LIN {X 0,Y 210.125,Z 422.294,A -85,B 0,C 180,E1 -20903.58,E2 -20903.58} C_VEL
LIN {X 0,Y 207.725,Z 422.606,A -85,B 0,C 180,E1 -20905.677,E2 -20905.677} C_VEL
LIN {X 0,Y 206.757,Z 422.716,A -85,B 0,C 180,E1 -20907.307,E2 -20907.307} C_VEL
LIN {X 0,Y 206.709,Z 422.715,A -85,B 0,C 180,E1 -20907.858,E2 -20907.858} C_VEL
LIN {X 0,Y 206.696,Z 422.724,A -85,B 0,C 180,E1 -20912.958,E2 -20912.958} C_VEL
LIN {X 0,Y 206.724,Z 422.922,A -85,B 0,C 180,E1 -20915.32,E2 -20915.32} C_VEL
LIN {X 0,Y 206.934,Z 423.791,A -85,B 0,C 180,E1 -20915.862,E2 -20915.862} C_VEL
LIN {X 0,Y 207.388,Z 425.01,A -85,B 0,C 180,E1 -20916.372,E2 -20916.372} C_VEL
LIN {X 0,Y 209.51,Z 427.919,A -85,B 0,C 180,E1 -20917.883,E2 -20917.883} C_VEL
LIN {X 0,Y 211.221,Z 431.051,A -85,B 0,C 180,E1 -20919.212,E2 -20919.212} C_VEL
LIN {X 0,Y 211.934,Z 431.967,A -85,B 0,C 180,E1 -20919.67,E2 -20919.67} C_VEL
LIN {X 0,Y 217.278,Z 441.785,A -85,B 0,C 180,E1 -20923.342,E2 -20923.342} C_VEL
LIN {X 0,Y 222.7,Z 451.851,A -85,B 0,C 180,E1 -20926.539,E2 -20926.539} C_VEL
LIN {X 0,Y 223.952,Z 454.762,A -85,B 0,C 180,E1 -20927.32,E2 -20927.32} C_VEL
LIN {X 0,Y 227.39,Z 471.394,A -85,B 0,C 180,E1 -20930.595,E2 -20930.595} C_VEL
LIN {X 0,Y 227.539,Z 474.416,A -85,B 0,C 180,E1 -20931.074,E2 -20931.074} C_VEL
LIN {X 0,Y 226.465,Z 488.855,A -85,B 0,C 180,E1 -20932.939,E2 -20932.939} C_VEL
LIN {X 0,Y 229.261,Z 519.875,A -85,B 0,C 180,E1 -20934.642,E2 -20934.642} C_VEL
LIN {X 0,Y 230.377,Z 537.62,A -85,B 0,C 180,E1 -20935.498,E2 -20935.498} C_VEL
LIN {X 0,Y 227.64,Z 600.474,A -85,B 0,C 180,E1 -20937.362,E2 -20937.362} C_VEL
LIN {X 0,Y 226.564,Z 613.93,A -85,B 0,C 180,E1 -20937.977,E2 -20937.977} C_VEL
LIN {X 0,Y 224.9,Z 626.109,A -85,B 0,C 180,E1 -20938.83,E2 -20938.83} C_VEL
LIN {X 0,Y 222.978,Z 637.557,A -85,B 0,C 180,E1 -20939.976,E2 -20939.976} C_VEL
LIN {X 0,Y 220.64,Z 648.728,A -85,B 0,C 180,E1 -20941.458,E2 -20941.458} C_VEL
LIN {X 0,Y 217.804,Z 660.086,A -85,B 0,C 180,E1 -20943.403,E2 -20943.403} C_VEL
LIN {X 0,Y 215.262,Z 669.231,A -85,B 0,C 180,E1 -20945.4,E2 -20945.4} C_VEL
LIN {X 0,Y 212.776,Z 678.047,A -85,B 0,C 180,E1 -20947.847,E2 -20947.847} C_VEL
LIN {X 0,Y 210.351,Z 685.667,A -85,B 0,C 180,E1 -20950.481,E2 -20950.481} C_VEL
LIN {X 0,Y 208.205,Z 692.195,A -85,B 0,C 180,E1 -20953.326,E2 -20953.326} C_VEL
LIN {X 0,Y 206.629,Z 697.379,A -85,B 0,C 180,E1 -20956.226,E2 -20956.226} C_VEL
LIN {X 0,Y 205.499,Z 701.381,A -85,B 0,C 180,E1 -20959.158,E2 -20959.158} C_VEL
LIN {X 0,Y 204.766,Z 704.328,A -85,B 0,C 180,E1 -20962.109,E2 -20962.109} C_VEL
LIN {X 0,Y 204.411,Z 706.558,A -85,B 0,C 180,E1 -20965.613,E2 -20965.613} C_VEL
LIN {X 0,Y 204.367,Z 707.347,A -85,B 0,C 180,E1 -20968.029,E2 -20968.029} C_VEL
LIN {X 0,Y 204.421,Z 707.561,A -85,B 0,C 180,E1 -20970,E2 -20970} C_VEL
LIN {X 0,Y 204.394,Z 707.335,A -85,B 0,C 180,E1 -20971.97,E2 -20971.97} C_VEL
LIN {X 0,Y 204.439,Z 706.499,A -85,B 0,C 180,E1 -20974.487,E2 -20974.487} C_VEL
LIN {X 0,Y 204.77,Z 704.285,A -85,B 0,C 180,E1 -20977.891,E2 -20977.891} C_VEL
LIN {X 0,Y 205.5,Z 701.321,A -85,B 0,C 180,E1 -20980.842,E2 -20980.842} C_VEL
LIN {X 0,Y 206.632,Z 697.298,A -85,B 0,C 180,E1 -20983.773,E2 -20983.773} C_VEL
LIN {X 0,Y 208.571,Z 691.095,A -85,B 0,C 180,E1 -20987.148,E2 -20987.148} C_VEL
LIN {X 0,Y 210.742,Z 684.327,A -85,B 0,C 180,E1 -20989.988,E2 -20989.988} C_VEL
LIN {X 0,Y 213.138,Z 676.486,A -85,B 0,C 180,E1 -20992.591,E2 -20992.591} C_VEL
LIN {X 0,Y 215.796,Z 667.107,A -85,B 0,C 180,E1 -20995.048,E2 -20995.048} C_VEL
LIN {X 0,Y 218.722,Z 656.357,A -85,B 0,C 180,E1 -20997.25,E2 -20997.25} C_VEL
LIN {X 0,Y 221.283,Z 645.5,A -85,B 0,C 180,E1 -20998.969,E2 -20998.969} C_VEL
LIN {X 0,Y 221.982,Z 642.83,A -85,B 0,C 180,E1 -20999.389,E2 -20999.389} C_VEL
LIN {X 0,Y 227.16,Z 636.768,A -85,B 0,C 180,E1 -21001.732,E2 -21001.732} C_VEL
LIN {X 0,Y 234.125,Z 628.278,A -85,B 0,C 180,E1 -21004.252,E2 -21004.252} C_VEL
LIN {X 0,Y 241.939,Z 617.995,A -85,B 0,C 180,E1 -21006.548,E2 -21006.548} C_VEL
LIN {X 0,Y 249.222,Z 607.391,A -85,B 0,C 180,E1 -21008.345,E2 -21008.345} C_VEL
LIN {X 0,Y 256.826,Z 594.892,A -85,B 0,C 180,E1 -21009.985,E2 -21009.985} C_VEL
LIN {X 0,Y 263.198,Z 583.1,A -85,B 0,C 180,E1 -21011.138,E2 -21011.138} C_VEL
LIN {X 0,Y 269.507,Z 569.488,A -85,B 0,C 180,E1 -21012.182,E2 -21012.182} C_VEL
LIN {X 0,Y 274.93,Z 555.525,A -85,B 0,C 180,E1 -21013.012,E2 -21013.012} C_VEL
LIN {X 0,Y 278.395,Z 544.603,A -85,B 0,C 180,E1 -21013.614,E2 -21013.614} C_VEL
LIN {X 0,Y 280.825,Z 534.789,A -85,B 0,C 180,E1 -21014.437,E2 -21014.437} C_VEL
LIN {X 0,Y 283.081,Z 524.784,A -85,B 0,C 180,E1 -21015.548,E2 -21015.548} C_VEL
LIN {X 0,Y 283.658,Z 522.171,A -85,B 0,C 180,E1 -21017.163,E2 -21017.163} C_VEL
LIN {X 0,Y 284.036,Z 521.4,A -85,B 0,C 180,E1 -21018.01,E2 -21018.01} C_VEL
LIN {X 0,Y 280.282,Z 536.18,A -85,B 0,C 180,E1 -21018.966,E2 -21018.966} C_VEL
LIN {X 0,Y 276.118,Z 548.931,A -85,B 0,C 180,E1 -21020.007,E2 -21020.007} C_VEL
LIN {X 0,Y 271.63,Z 559.907,A -85,B 0,C 180,E1 -21021.139,E2 -21021.139} C_VEL
LIN {X 0,Y 266.158,Z 571.085,A -85,B 0,C 180,E1 -21022.604,E2 -21022.604} C_VEL
LIN {X 0,Y 259.706,Z 582.081,A -85,B 0,C 180,E1 -21024.421,E2 -21024.421} C_VEL
LIN {X 0,Y 253.474,Z 591.011,A -85,B 0,C 180,E1 -21026.321,E2 -21026.321} C_VEL
LIN {X 0,Y 247.643,Z 598.282,A -85,B 0,C 180,E1 -21028.33,E2 -21028.33} C_VEL
LIN {X 0,Y 242.063,Z 604.273,A -85,B 0,C 180,E1 -21030.424,E2 -21030.424} C_VEL
LIN {X 0,Y 236.808,Z 609.042,A -85,B 0,C 180,E1 -21032.612,E2 -21032.612} C_VEL
LIN {X 0,Y 231.875,Z 612.783,A -85,B 0,C 180,E1 -21034.892,E2 -21034.892} C_VEL
LIN {X 0,Y 228.801,Z 614.725,A -85,B 0,C 180,E1 -21036.465,E2 -21036.465} C_VEL
LIN {X 0,Y 225.905,Z 616.243,A -85,B 0,C 180,E1 -21038.079,E2 -21038.079} C_VEL
LIN {X 0,Y 220.673,Z 618.05,A -85,B 0,C 180,E1 -21041.429,E2 -21041.429} C_VEL
LIN {X 0,Y 216.251,Z 618.267,A -85,B 0,C 180,E1 -21044.93,E2 -21044.93} C_VEL
LIN {X 0,Y 214.361,Z 617.789,A -85,B 0,C 180,E1 -21046.732,E2 -21046.732} C_VEL
LIN {X 0,Y 211.13,Z 615.597,A -85,B 0,C 180,E1 -21050.419,E2 -21050.419} C_VEL
LIN {X 0,Y 209.081,Z 611.799,A -85,B 0,C 180,E1 -21054.212,E2 -21054.212} C_VEL
LIN {X 0,Y 207.793,Z 607.81,A -85,B 0,C 180,E1 -21057.092,E2 -21057.092} C_VEL
LIN {X 0,Y 206.849,Z 602.743,A -85,B 0,C 180,E1 -21060,E2 -21060} C_VEL
LIN {X 0,Y 206.563,Z 596.507,A -85,B 0,C 180,E1 -21062.925,E2 -21062.925} C_VEL
LIN {X 0,Y 206.557,Z 588.898,A -85,B 0,C 180,E1 -21065.859,E2 -21065.859} C_VEL
LIN {X 0,Y 207.079,Z 579.651,A -85,B 0,C 180,E1 -21068.785,E2 -21068.785} C_VEL
LIN {X 0,Y 207.718,Z 568.213,A -85,B 0,C 180,E1 -21071.713,E2 -21071.713} C_VEL
LIN {X 0,Y 208.439,Z 556.478,A -85,B 0,C 180,E1 -21074.15,E2 -21074.15} C_VEL
LIN {X 0,Y 209.247,Z 543.434,A -85,B 0,C 180,E1 -21076.337,E2 -21076.337} C_VEL
LIN {X 0,Y 210.03,Z 530.574,A -85,B 0,C 180,E1 -21078.031,E2 -21078.031} C_VEL
LIN {X 0,Y 210.712,Z 517.623,A -85,B 0,C 180,E1 -21079.357,E2 -21079.357} C_VEL
LIN {X 0,Y 211.208,Z 501.844,A -85,B 0,C 180,E1 -21080.514,E2 -21080.514} C_VEL
LIN {X 0,Y 212.82,Z 450.947,A -85,B 0,C 180,E1 -21083.43,E2 -21083.43} C_VEL
LIN {X 0,Y 212.897,Z 445.737,A -85,B 0,C 180,E1 -21083.732,E2 -21083.732} C_VEL
LIN {X 0,Y 207.049,Z 423.827,A -85,B 0,C 180,E1 -21085.256,E2 -21085.256} C_VEL
LIN {X 0,Y 206.827,Z 422.814,A -85,B 0,C 180,E1 -21085.631,E2 -21085.631} C_VEL
LIN {X 0,Y 206.74,Z 422.955,A -85,B 0,C 180,E1 -21088.558,E2 -21088.558} C_VEL
LIN {X 0,Y 207.205,Z 424.593,A -85,B 0,C 180,E1 -21089.46,E2 -21089.46} C_VEL
LIN {X 0,Y 209.921,Z 429.877,A -85,B 0,C 180,E1 -21092.389,E2 -21092.389} C_VEL
LIN {X 0,Y 212.673,Z 435.853,A -85,B 0,C 180,E1 -21095.332,E2 -21095.332} C_VEL
LIN {X 0,Y 215.756,Z 443.211,A -85,B 0,C 180,E1 -21098.577,E2 -21098.577} C_VEL
LIN {X 0,Y 219.359,Z 453.452,A -85,B 0,C 180,E1 -21102.533,E2 -21102.533} C_VEL
LIN {X 0,Y 222.064,Z 462.255,A -85,B 0,C 180,E1 -21105.6,E2 -21105.6} C_VEL
LIN {X 0,Y 224.578,Z 472.081,A -85,B 0,C 180,E1 -21108.683,E2 -21108.683} C_VEL
LIN {X 0,Y 226.464,Z 481.184,A -85,B 0,C 180,E1 -21111.287,E2 -21111.287} C_VEL
LIN {X 0,Y 226.441,Z 483.891,A -85,B 0,C 180,E1 -21111.913,E2 -21111.913} C_VEL
LIN {X 0,Y 225.76,Z 488.467,A -85,B 0,C 180,E1 -21112.757,E2 -21112.757} C_VEL
LIN {X 0,Y 229.102,Z 514.329,A -85,B 0,C 180,E1 -21114.381,E2 -21114.381} C_VEL
LIN {X 0,Y 230.932,Z 531.932,A -85,B 0,C 180,E1 -21115.361,E2 -21115.361} C_VEL
LIN {X 0,Y 227.845,Z 601.159,A -85,B 0,C 180,E1 -21117.461,E2 -21117.461} C_VEL
LIN {X 0,Y 226.566,Z 613.791,A -85,B 0,C 180,E1 -21118.109,E2 -21118.109} C_VEL
LIN {X 0,Y 224.871,Z 626.008,A -85,B 0,C 180,E1 -21119.088,E2 -21119.088} C_VEL
LIN {X 0,Y 222.676,Z 638.356,A -85,B 0,C 180,E1 -21120.452,E2 -21120.452} C_VEL
LIN {X 0,Y 220.334,Z 648.71,A -85,B 0,C 180,E1 -21121.935,E2 -21121.935} C_VEL
LIN {X 0,Y 217.622,Z 659.321,A -85,B 0,C 180,E1 -21123.895,E2 -21123.895} C_VEL
LIN {X 0,Y 214.928,Z 669.044,A -85,B 0,C 180,E1 -21126.183,E2 -21126.183} C_VEL
LIN {X 0,Y 212.411,Z 677.426,A -85,B 0,C 180,E1 -21128.657,E2 -21128.657} C_VEL
LIN {X 0,Y 210.005,Z 684.913,A -85,B 0,C 180,E1 -21131.463,E2 -21131.463} C_VEL
LIN {X 0,Y 207.957,Z 690.92,A -85,B 0,C 180,E1 -21134.314,E2 -21134.314} C_VEL
LIN {X 0,Y 206.472,Z 695.67,A -85,B 0,C 180,E1 -21137.218,E2 -21137.218} C_VEL
LIN {X 0,Y 205.439,Z 699.303,A -85,B 0,C 180,E1 -21140.151,E2 -21140.151} C_VEL
LIN {X 0,Y 204.934,Z 701.174,A -85,B 0,C 180,E1 -21142.116,E2 -21142.116} C_VEL
LIN {X 0,Y 204.412,Z 703.421,A -85,B 0,C 180,E1 -21145.613,E2 -21145.613} C_VEL
LIN {X 0,Y 204.318,Z 704.213,A -85,B 0,C 180,E1 -21148.029,E2 -21148.029} C_VEL
LIN {X 0,Y 204.344,Z 704.445,A -85,B 0,C 180,E1 -21150,E2 -21150} C_VEL
LIN {X 0,Y 204.318,Z 704.247,A -85,B 0,C 180,E1 -21151.971,E2 -21151.971} C_VEL
LIN {X 0,Y 204.422,Z 703.462,A -85,B 0,C 180,E1 -21154.423,E2 -21154.423} C_VEL
LIN {X 0,Y 204.873,Z 701.295,A -85,B 0,C 180,E1 -21157.887,E2 -21157.887} C_VEL
LIN {X 0,Y 205.702,Z 698.396,A -85,B 0,C 180,E1 -21160.831,E2 -21160.831} C_VEL
LIN {X 0,Y 206.868,Z 694.457,A -85,B 0,C 180,E1 -21163.758,E2 -21163.758} C_VEL
LIN {X 0,Y 208.521,Z 689.352,A -85,B 0,C 180,E1 -21166.648,E2 -21166.648} C_VEL
LIN {X 0,Y 210.727,Z 682.917,A -85,B 0,C 180,E1 -21169.483,E2 -21169.483} C_VEL
LIN {X 0,Y 213.184,Z 675.164,A -85,B 0,C 180,E1 -21172.195,E2 -21172.195} C_VEL
LIN {X 0,Y 215.627,Z 666.748,A -85,B 0,C 180,E1 -21174.555,E2 -21174.555} C_VEL
LIN {X 0,Y 218.371,Z 656.669,A -85,B 0,C 180,E1 -21176.781,E2 -21176.781} C_VEL
LIN {X 0,Y 221.228,Z 645.334,A -85,B 0,C 180,E1 -21178.718,E2 -21178.718} C_VEL
LIN {X 0,Y 223.562,Z 634.155,A -85,B 0,C 180,E1 -21180.198,E2 -21180.198} C_VEL
LIN {X 0,Y 225.627,Z 621.463,A -85,B 0,C 180,E1 -21181.45,E2 -21181.45} C_VEL
LIN {X 0,Y 227.26,Z 608.917,A -85,B 0,C 180,E1 -21182.305,E2 -21182.305} C_VEL
LIN {X 0,Y 228.292,Z 595.778,A -85,B 0,C 180,E1 -21182.86,E2 -21182.86} C_VEL
LIN {X 0,Y 230.95,Z 530.487,A -85,B 0,C 180,E1 -21184.837,E2 -21184.837} C_VEL
LIN {X 0,Y 227.386,Z 499.475,A -85,B 0,C 180,E1 -21186.651,E2 -21186.651} C_VEL
LIN {X 0,Y 225.832,Z 487.938,A -85,B 0,C 180,E1 -21187.431,E2 -21187.431} C_VEL
LIN {X 0,Y 226.543,Z 483.152,A -85,B 0,C 180,E1 -21188.35,E2 -21188.35} C_VEL
LIN {X 0,Y 226.144,Z 479.35,A -85,B 0,C 180,E1 -21189.371,E2 -21189.371} C_VEL
LIN {X 0,Y 223.963,Z 469.191,A -85,B 0,C 180,E1 -21192.334,E2 -21192.334} C_VEL
LIN {X 0,Y 221.211,Z 459.114,A -85,B 0,C 180,E1 -21195.657,E2 -21195.657} C_VEL
LIN {X 0,Y 217.494,Z 447.851,A -85,B 0,C 180,E1 -21199.739,E2 -21199.739} C_VEL
LIN {X 0,Y 213.697,Z 438.3,A -85,B 0,C 180,E1 -21203.702,E2 -21203.702} C_VEL
LIN {X 0,Y 210.588,Z 431.05,A -85,B 0,C 180,E1 -21207.158,E2 -21207.158} C_VEL
LIN {X 0,Y 208.37,Z 426.435,A -85,B 0,C 180,E1 -21209.607,E2 -21209.607} C_VEL
LIN {X 0,Y 206.831,Z 423.491,A -85,B 0,C 180,E1 -21211.317,E2 -21211.317} C_VEL
LIN {X 0,Y 206.717,Z 422.755,A -85,B 0,C 180,E1 -21211.945,E2 -21211.945} C_VEL
LIN {X 0,Y 206.74,Z 422.709,A -85,B 0,C 180,E1 -21216.615,E2 -21216.615} C_VEL
LIN {X 0,Y 206.805,Z 422.695,A -85,B 0,C 180,E1 -21222.19,E2 -21222.19} C_VEL
LIN {X 0,Y 206.858,Z 422.706,A -85,B 0,C 180,E1 -21226.242,E2 -21226.242} C_VEL
LIN {X 0,Y 207.081,Z 422.666,A -85,B 0,C 180,E1 -21230.23,E2 -21230.23} C_VEL
LIN {X 0,Y 207.04,Z 422.665,A -85,B 0,C 180,E1 -21234.155,E2 -21234.155} C_VEL
LIN {X 0,Y 207.346,Z 422.647,A -85,B 0,C 180,E1 -21238.057,E2 -21238.057} C_VEL
LIN {X 0,Y 207.483,Z 422.627,A -85,B 0,C 180,E1 -21240,E2 -21240} C_VEL
LIN {X 0,Y 207.344,Z 422.621,A -85,B 0,C 180,E1 -21241.942,E2 -21241.942} C_VEL
LIN {X 0,Y 207.125,Z 422.662,A -85,B 0,C 180,E1 -21247.8,E2 -21247.8} C_VEL
LIN {X 0,Y 206.905,Z 422.692,A -85,B 0,C 180,E1 -21251.759,E2 -21251.759} C_VEL
LIN {X 0,Y 206.802,Z 422.693,A -85,B 0,C 180,E1 -21255.776,E2 -21255.776} C_VEL
LIN {X 0,Y 206.713,Z 422.738,A -85,B 0,C 180,E1 -21259.876,E2 -21259.876} C_VEL
LIN {X 0,Y 206.693,Z 422.712,A -85,B 0,C 180,E1 -21264.081,E2 -21264.081} C_VEL
LIN {X 0,Y 206.709,Z 422.715,A -85,B 0,C 180,E1 -21267.858,E2 -21267.858} C_VEL
LIN {X 0,Y 205.999,Z 422.804,A -85,B 0,C 180,E1 -21268.977,E2 -21268.977} C_VEL
LIN {X 0,Y 202.98,Z 423.24,A -85,B 0,C 180,E1 -21270.734,E2 -21270.734} C_VEL
LIN {X 0,Y 200.627,Z 424.443,A -85,B 0,C 180,E1 -21272.296,E2 -21272.296} C_VEL
LIN {X 0,Y 200.311,Z 425.566,A -85,B 0,C 180,E1 -21273.175,E2 -21273.175} C_VEL
LIN {X 0,Y 200.527,Z 426.115,A -85,B 0,C 180,E1 -21273.51,E2 -21273.51} C_VEL
LIN {X 0,Y 202.62,Z 428.995,A -85,B 0,C 180,E1 -21275.264,E2 -21275.264} C_VEL
LIN {X 0,Y 203.311,Z 430.638,A -85,B 0,C 180,E1 -21275.991,E2 -21275.991} C_VEL
LIN {X 0,Y 205.235,Z 433.407,A -85,B 0,C 180,E1 -21277.433,E2 -21277.433} C_VEL
LIN {X 0,Y 211.094,Z 443.839,A -85,B 0,C 180,E1 -21281.749,E2 -21281.749} C_VEL
LIN {X 0,Y 216.926,Z 454.828,A -85,B 0,C 180,E1 -21285.46,E2 -21285.46} C_VEL
LIN {X 0,Y 218.761,Z 458.802,A -85,B 0,C 180,E1 -21286.623,E2 -21286.623} C_VEL
LIN {X 0,Y 221.749,Z 474.672,A -85,B 0,C 180,E1 -21289.872,E2 -21289.872} C_VEL
LIN {X 0,Y 220.723,Z 488.982,A -85,B 0,C 180,E1 -21291.807,E2 -21291.807} C_VEL
LIN {X 0,Y 223.416,Z 519.627,A -85,B 0,C 180,E1 -21293.559,E2 -21293.559} C_VEL
LIN {X 0,Y 224.571,Z 537.268,A -85,B 0,C 180,E1 -21294.457,E2 -21294.457} C_VEL
LIN {X 0,Y 221.714,Z 600.522,A -85,B 0,C 180,E1 -21296.376,E2 -21296.376} C_VEL
LIN {X 0,Y 220.585,Z 613.934,A -85,B 0,C 180,E1 -21297.001,E2 -21297.001} C_VEL
LIN {X 0,Y 218.869,Z 626.093,A -85,B 0,C 180,E1 -21297.87,E2 -21297.87} C_VEL
LIN {X 0,Y 216.86,Z 637.527,A -85,B 0,C 180,E1 -21299.037,E2 -21299.037} C_VEL
LIN {X 0,Y 214.425,Z 648.691,A -85,B 0,C 180,E1 -21300.551,E2 -21300.551} C_VEL
LIN {X 0,Y 211.472,Z 660.045,A -85,B 0,C 180,E1 -21302.54,E2 -21302.54} C_VEL
LIN {X 0,Y 208.813,Z 669.186,A -85,B 0,C 180,E1 -21304.588,E2 -21304.588} C_VEL
LIN {X 0,Y 206.019,Z 678.572,A -85,B 0,C 180,E1 -21307.287,E2 -21307.287} C_VEL
LIN {X 0,Y 203.64,Z 685.617,A -85,B 0,C 180,E1 -21309.81,E2 -21309.81} C_VEL
LIN {X 0,Y 201.41,Z 692.144,A -85,B 0,C 180,E1 -21312.746,E2 -21312.746} C_VEL
LIN {X 0,Y 199.692,Z 697.327,A -85,B 0,C 180,E1 -21315.737,E2 -21315.737} C_VEL
LIN {X 0,Y 198.521,Z 701.328,A -85,B 0,C 180,E1 -21318.772,E2 -21318.772} C_VEL
LIN {X 0,Y 197.717,Z 704.275,A -85,B 0,C 180,E1 -21321.825,E2 -21321.825} C_VEL
LIN {X 0,Y 197.338,Z 706.604,A -85,B 0,C 180,E1 -21325.708,E2 -21325.708} C_VEL
LIN {X 0,Y 197.275,Z 707.293,A -85,B 0,C 180,E1 -21327.958,E2 -21327.958} C_VEL
LIN {X 0,Y 197.325,Z 707.507,A -85,B 0,C 180,E1 -21330,E2 -21330} C_VEL
LIN {X 0,Y 197.302,Z 707.281,A -85,B 0,C 180,E1 -21332.041,E2 -21332.041} C_VEL
LIN {X 0,Y 197.338,Z 706.584,A -85,B 0,C 180,E1 -21334.291,E2 -21334.291} C_VEL
LIN {X 0,Y 197.72,Z 704.231,A -85,B 0,C 180,E1 -21338.174,E2 -21338.174} C_VEL
LIN {X 0,Y 198.523,Z 701.267,A -85,B 0,C 180,E1 -21341.227,E2 -21341.227} C_VEL
LIN {X 0,Y 199.695,Z 697.243,A -85,B 0,C 180,E1 -21344.262,E2 -21344.262} C_VEL
LIN {X 0,Y 201.786,Z 691.041,A -85,B 0,C 180,E1 -21347.743,E2 -21347.743} C_VEL
LIN {X 0,Y 204.036,Z 684.274,A -85,B 0,C 180,E1 -21350.674,E2 -21350.674} C_VEL
LIN {X 0,Y 206.362,Z 677.111,A -85,B 0,C 180,E1 -21353.142,E2 -21353.142} C_VEL
LIN {X 0,Y 208.805,Z 668.98,A -85,B 0,C 180,E1 -21355.413,E2 -21355.413} C_VEL
LIN {X 0,Y 211.786,Z 658.631,A -85,B 0,C 180,E1 -21357.683,E2 -21357.683} C_VEL
LIN {X 0,Y 214.43,Z 648.387,A -85,B 0,C 180,E1 -21359.448,E2 -21359.448} C_VEL
LIN {X 0,Y 215.636,Z 643.568,A -85,B 0,C 180,E1 -21360.208,E2 -21360.208} C_VEL
LIN {X 0,Y 222.196,Z 636.688,A -85,B 0,C 180,E1 -21363.066,E2 -21363.066} C_VEL
LIN {X 0,Y 228.367,Z 629.883,A -85,B 0,C 180,E1 -21365.242,E2 -21365.242} C_VEL
LIN {X 0,Y 236.374,Z 620.396,A -85,B 0,C 180,E1 -21367.555,E2 -21367.555} C_VEL
LIN {X 0,Y 243.798,Z 610.687,A -85,B 0,C 180,E1 -21369.36,E2 -21369.36} C_VEL
LIN {X 0,Y 251.591,Z 599.26,A -85,B 0,C 180,E1 -21370.992,E2 -21370.992} C_VEL
LIN {X 0,Y 258.67,Z 587.621,A -85,B 0,C 180,E1 -21372.257,E2 -21372.257} C_VEL
LIN {X 0,Y 265.941,Z 573.767,A -85,B 0,C 180,E1 -21373.401,E2 -21373.401} C_VEL
LIN {X 0,Y 271.955,Z 560.246,A -85,B 0,C 180,E1 -21374.247,E2 -21374.247} C_VEL
LIN {X 0,Y 276.893,Z 546.691,A -85,B 0,C 180,E1 -21374.977,E2 -21374.977} C_VEL
LIN {X 0,Y 279.807,Z 536.743,A -85,B 0,C 180,E1 -21375.828,E2 -21375.828} C_VEL
LIN {X 0,Y 281.526,Z 530.217,A -85,B 0,C 180,E1 -21376.577,E2 -21376.577} C_VEL
LIN {X 0,Y 281.704,Z 529.57,A -85,B 0,C 180,E1 -21376.977,E2 -21376.977} C_VEL
LIN {X 0,Y 277.359,Z 544.079,A -85,B 0,C 180,E1 -21378.029,E2 -21378.029} C_VEL
LIN {X 0,Y 271.937,Z 557.756,A -85,B 0,C 180,E1 -21379.264,E2 -21379.264} C_VEL
LIN {X 0,Y 266.162,Z 569.466,A -85,B 0,C 180,E1 -21380.675,E2 -21380.675} C_VEL
LIN {X 0,Y 260.442,Z 579.207,A -85,B 0,C 180,E1 -21382.127,E2 -21382.127} C_VEL
LIN {X 0,Y 253.944,Z 588.605,A -85,B 0,C 180,E1 -21383.887,E2 -21383.887} C_VEL
LIN {X 0,Y 247.351,Z 596.783,A -85,B 0,C 180,E1 -21385.864,E2 -21385.864} C_VEL
LIN {X 0,Y 242.289,Z 602.24,A -85,B 0,C 180,E1 -21387.546,E2 -21387.546} C_VEL
LIN {X 0,Y 236.494,Z 607.683,A -85,B 0,C 180,E1 -21389.656,E2 -21389.656} C_VEL
LIN {X 0,Y 231.191,Z 611.929,A -85,B 0,C 180,E1 -21391.79,E2 -21391.79} C_VEL
LIN {X 0,Y 225.863,Z 615.396,A -85,B 0,C 180,E1 -21394.175,E2 -21394.175} C_VEL
LIN {X 0,Y 219.626,Z 618.364,A -85,B 0,C 180,E1 -21397.418,E2 -21397.418} C_VEL
LIN {X 0,Y 214.15,Z 619.742,A -85,B 0,C 180,E1 -21400.842,E2 -21400.842} C_VEL
LIN {X 0,Y 209.527,Z 619.53,A -85,B 0,C 180,E1 -21404.435,E2 -21404.435} C_VEL
LIN {X 0,Y 205.743,Z 617.761,A -85,B 0,C 180,E1 -21408.173,E2 -21408.173} C_VEL
LIN {X 0,Y 204.191,Z 616.283,A -85,B 0,C 180,E1 -21410.09,E2 -21410.09} C_VEL
LIN {X 0,Y 202.038,Z 612.043,A -85,B 0,C 180,E1 -21414.01,E2 -21414.01} C_VEL
LIN {X 0,Y 200.711,Z 607.763,A -85,B 0,C 180,E1 -21416.989,E2 -21416.989} C_VEL
LIN {X 0,Y 199.716,Z 601.389,A -85,B 0,C 180,E1 -21420.504,E2 -21420.504} C_VEL
LIN {X 0,Y 199.453,Z 594.548,A -85,B 0,C 180,E1 -21423.535,E2 -21423.535} C_VEL
LIN {X 0,Y 199.562,Z 586.272,A -85,B 0,C 180,E1 -21426.572,E2 -21426.572} C_VEL
LIN {X 0,Y 200.035,Z 578.078,A -85,B 0,C 180,E1 -21429.097,E2 -21429.097} C_VEL
LIN {X 0,Y 200.676,Z 567.159,A -85,B 0,C 180,E1 -21431.865,E2 -21431.865} C_VEL
LIN {X 0,Y 201.43,Z 554.863,A -85,B 0,C 180,E1 -21434.395,E2 -21434.395} C_VEL
LIN {X 0,Y 202.184,Z 542.752,A -85,B 0,C 180,E1 -21436.405,E2 -21436.405} C_VEL
LIN {X 0,Y 203.083,Z 528.53,A -85,B 0,C 180,E1 -21438.278,E2 -21438.278} C_VEL
LIN {X 0,Y 203.734,Z 514.657,A -85,B 0,C 180,E1 -21439.654,E2 -21439.654} C_VEL
LIN {X 0,Y 204.167,Z 498.753,A -85,B 0,C 180,E1 -21440.776,E2 -21440.776} C_VEL
LIN {X 0,Y 205.842,Z 446.863,A -85,B 0,C 180,E1 -21443.883,E2 -21443.883} C_VEL
LIN {X 0,Y 200.267,Z 425.798,A -85,B 0,C 180,E1 -21445.406,E2 -21445.406} C_VEL
LIN {X 0,Y 199.955,Z 424.631,A -85,B 0,C 180,E1 -21445.782,E2 -21445.782} C_VEL
LIN {X 0,Y 200.098,Z 424.985,A -85,B 0,C 180,E1 -21446.322,E2 -21446.322} C_VEL
LIN {X 0,Y 203.305,Z 431.331,A -85,B 0,C 180,E1 -21450.206,E2 -21450.206} C_VEL
LIN {X 0,Y 206.949,Z 439.285,A -85,B 0,C 180,E1 -21454.432,E2 -21454.432} C_VEL
LIN {X 0,Y 210.337,Z 447.557,A -85,B 0,C 180,E1 -21458.181,E2 -21458.181} C_VEL
LIN {X 0,Y 213.448,Z 456.635,A -85,B 0,C 180,E1 -21461.817,E2 -21461.817} C_VEL
LIN {X 0,Y 216.031,Z 465.063,A -85,B 0,C 180,E1 -21464.848,E2 -21464.848} C_VEL
LIN {X 0,Y 218.319,Z 474.035,A -85,B 0,C 180,E1 -21467.766,E2 -21467.766} C_VEL
LIN {X 0,Y 220.348,Z 483.903,A -85,B 0,C 180,E1 -21470.664,E2 -21470.664} C_VEL
LIN {X 0,Y 220.24,Z 486.308,A -85,B 0,C 180,E1 -21471.223,E2 -21471.223} C_VEL
LIN {X 0,Y 219.971,Z 488.474,A -85,B 0,C 180,E1 -21471.604,E2 -21471.604} C_VEL
LIN {X 0,Y 223.244,Z 514.292,A -85,B 0,C 180,E1 -21473.297,E2 -21473.297} C_VEL
LIN {X 0,Y 225.094,Z 531.875,A -85,B 0,C 180,E1 -21474.327,E2 -21474.327} C_VEL
LIN {X 0,Y 221.913,Z 601.152,A -85,B 0,C 180,E1 -21476.479,E2 -21476.479} C_VEL
LIN {X 0,Y 220.575,Z 613.815,A -85,B 0,C 180,E1 -21477.136,E2 -21477.136} C_VEL
LIN {X 0,Y 218.819,Z 626.044,A -85,B 0,C 180,E1 -21478.134,E2 -21478.134} C_VEL
LIN {X 0,Y 216.527,Z 638.398,A -85,B 0,C 180,E1 -21479.526,E2 -21479.526} C_VEL
LIN {X 0,Y 214.099,Z 648.757,A -85,B 0,C 180,E1 -21481.041,E2 -21481.041} C_VEL
LIN {X 0,Y 211.244,Z 659.371,A -85,B 0,C 180,E1 -21483.045,E2 -21483.045} C_VEL
LIN {X 0,Y 208.765,Z 668.048,A -85,B 0,C 180,E1 -21485.116,E2 -21485.116} C_VEL
LIN {X 0,Y 206.233,Z 676.144,A -85,B 0,C 180,E1 -21487.5,E2 -21487.5} C_VEL
LIN {X 0,Y 203.651,Z 683.846,A -85,B 0,C 180,E1 -21490.338,E2 -21490.338} C_VEL
LIN {X 0,Y 201.785,Z 689.129,A -85,B 0,C 180,E1 -21492.78,E2 -21492.78} C_VEL
LIN {X 0,Y 200.037,Z 694.29,A -85,B 0,C 180,E1 -21495.763,E2 -21495.763} C_VEL
LIN {X 0,Y 198.762,Z 698.284,A -85,B 0,C 180,E1 -21498.786,E2 -21498.786} C_VEL
LIN {X 0,Y 197.905,Z 701.228,A -85,B 0,C 180,E1 -21501.834,E2 -21501.834} C_VEL
LIN {X 0,Y 197.516,Z 702.653,A -85,B 0,C 180,E1 -21503.872,E2 -21503.872} C_VEL
LIN {X 0,Y 197.326,Z 703.652,A -85,B 0,C 180,E1 -21505.915,E2 -21505.915} C_VEL
LIN {X 0,Y 197.231,Z 704.267,A -85,B 0,C 180,E1 -21507.958,E2 -21507.958} C_VEL
LIN {X 0,Y 197.251,Z 704.499,A -85,B 0,C 180,E1 -21510,E2 -21510} C_VEL
LIN {X 0,Y 197.23,Z 704.3,A -85,B 0,C 180,E1 -21512.042,E2 -21512.042} C_VEL
LIN {X 0,Y 197.344,Z 703.618,A -85,B 0,C 180,E1 -21514.314,E2 -21514.314} C_VEL
LIN {X 0,Y 197.822,Z 701.348,A -85,B 0,C 180,E1 -21518.17,E2 -21518.17} C_VEL
LIN {X 0,Y 198.704,Z 698.448,A -85,B 0,C 180,E1 -21521.218,E2 -21521.218} C_VEL
LIN {X 0,Y 199.976,Z 694.508,A -85,B 0,C 180,E1 -21524.242,E2 -21524.242} C_VEL
LIN {X 0,Y 201.701,Z 689.402,A -85,B 0,C 180,E1 -21527.228,E2 -21527.228} C_VEL
LIN {X 0,Y 204.036,Z 682.966,A -85,B 0,C 180,E1 -21530.149,E2 -21530.149} C_VEL
LIN {X 0,Y 206.52,Z 675.52,A -85,B 0,C 180,E1 -21532.839,E2 -21532.839} C_VEL
LIN {X 0,Y 209.162,Z 666.792,A -85,B 0,C 180,E1 -21535.367,E2 -21535.367} C_VEL
LIN {X 0,Y 212.077,Z 656.709,A -85,B 0,C 180,E1 -21537.642,E2 -21537.642} C_VEL
LIN {X 0,Y 215.027,Z 645.371,A -85,B 0,C 180,E1 -21539.627,E2 -21539.627} C_VEL
LIN {X 0,Y 217.45,Z 634.183,A -85,B 0,C 180,E1 -21541.14,E2 -21541.14} C_VEL
LIN {X 0,Y 219.62,Z 621.479,A -85,B 0,C 180,E1 -21542.413,E2 -21542.413} C_VEL
LIN {X 0,Y 221.301,Z 608.913,A -85,B 0,C 180,E1 -21543.286,E2 -21543.286} C_VEL
LIN {X 0,Y 222.378,Z 595.71,A -85,B 0,C 180,E1 -21543.85,E2 -21543.85} C_VEL
LIN {X 0,Y 225.119,Z 531.275,A -85,B 0,C 180,E1 -21545.843,E2 -21545.843} C_VEL
LIN {X 0,Y 221.841,Z 501.831,A -85,B 0,C 180,E1 -21547.626,E2 -21547.626} C_VEL
LIN {X 0,Y 220.034,Z 487.884,A -85,B 0,C 180,E1 -21548.602,E2 -21548.602} C_VEL
LIN {X 0,Y 220.421,Z 484.262,A -85,B 0,C 180,E1 -21549.359,E2 -21549.359} C_VEL
LIN {X 0,Y 218.266,Z 473.539,A -85,B 0,C 180,E1 -21552.547,E2 -21552.547} C_VEL
LIN {X 0,Y 215.316,Z 462.326,A -85,B 0,C 180,E1 -21556.31,E2 -21556.31} C_VEL
LIN {X 0,Y 211.736,Z 451.348,A -85,B 0,C 180,E1 -21560.443,E2 -21560.443} C_VEL
LIN {X 0,Y 208.565,Z 443.1,A -85,B 0,C 180,E1 -21563.973,E2 -21563.973} C_VEL
LIN {X 0,Y 205.159,Z 435.05,A -85,B 0,C 180,E1 -21567.928,E2 -21567.928} C_VEL
LIN {X 0,Y 201.583,Z 427.646,A -85,B 0,C 180,E1 -21572.118,E2 -21572.118} C_VEL
LIN {X 0,Y 199.986,Z 425.039,A -85,B 0,C 180,E1 -21573.942,E2 -21573.942} C_VEL
LIN {X 0,Y 199.651,Z 423.627,A -85,B 0,C 180,E1 -21575.013,E2 -21575.013} C_VEL
LIN {X 0,Y 199.649,Z 423.617,A -85,B 0,C 180,E1 -21579.389,E2 -21579.389} C_VEL
LIN {X 0,Y 199.747,Z 423.582,A -85,B 0,C 180,E1 -21583.651,E2 -21583.651} C_VEL
LIN {X 0,Y 199.856,Z 423.558,A -85,B 0,C 180,E1 -21587.819,E2 -21587.819} C_VEL
LIN {X 0,Y 200.078,Z 423.563,A -85,B 0,C 180,E1 -21591.923,E2 -21591.923} C_VEL
LIN {X 0,Y 200.288,Z 423.524,A -85,B 0,C 180,E1 -21597.989,E2 -21597.989} C_VEL
LIN {X 0,Y 200.45,Z 423.502,A -85,B 0,C 180,E1 -21600,E2 -21600} C_VEL
LIN {X 0,Y 199.986,Z 423.544,A -85,B 0,C 180,E1 -21604.03,E2 -21604.03} C_VEL
LIN {X 0,Y 200.073,Z 423.536,A -85,B 0,C 180,E1 -21608.077,E2 -21608.077} C_VEL
LIN {X 0,Y 199.855,Z 423.577,A -85,B 0,C 180,E1 -21612.18,E2 -21612.18} C_VEL
LIN {X 0,Y 199.743,Z 423.569,A -85,B 0,C 180,E1 -21616.349,E2 -21616.349} C_VEL
LIN {X 0,Y 199.643,Z 423.609,A -85,B 0,C 180,E1 -21620.611,E2 -21620.611} C_VEL
LIN {X 0,Y 199.623,Z 423.602,A -85,B 0,C 180,E1 -21624.991,E2 -21624.991} C_VEL
LIN {X 0,Y 199.609,Z 423.594,A -85,B 0,C 180,E1 -21629.533,E2 -21629.533} C_VEL
LIN {X 0,Y 199.699,Z 423.777,A -85,B 0,C 180,E1 -21632.158,E2 -21632.158} C_VEL
LIN {X 0,Y 199.951,Z 424.935,A -85,B 0,C 180,E1 -21632.896,E2 -21632.896} C_VEL
LIN {X 0,Y 200.527,Z 426.115,A -85,B 0,C 180,E1 -21633.51,E2 -21633.51} C_VEL
LIN {X 0,Y 201.695,Z 429.264,A -85,B 0,C 180,E1 -21634.895,E2 -21634.895} C_VEL
LIN {X 0,Y 202.674,Z 435.958,A -85,B 0,C 180,E1 -21636.956,E2 -21636.956} C_VEL
LIN {X 0,Y 203.468,Z 441.587,A -85,B 0,C 180,E1 -21638.553,E2 -21638.553} C_VEL
LIN {X 0,Y 204.633,Z 445.375,A -85,B 0,C 180,E1 -21639.81,E2 -21639.81} C_VEL
LIN {X 0,Y 205.204,Z 446.47,A -85,B 0,C 180,E1 -21640.246,E2 -21640.246} C_VEL
LIN {X 0,Y 209.721,Z 454.949,A -85,B 0,C 180,E1 -21643.392,E2 -21643.392} C_VEL
LIN {X 0,Y 213.368,Z 462.241,A -85,B 0,C 180,E1 -21645.759,E2 -21645.759} C_VEL
LIN {X 0,Y 215.496,Z 474.082,A -85,B 0,C 180,E1 -21648.325,E2 -21648.325} C_VEL
LIN {X 0,Y 216.076,Z 477.552,A -85,B 0,C 180,E1 -21649.034,E2 -21649.034} C_VEL
LIN {X 0,Y 215.069,Z 489.064,A -85,B 0,C 180,E1 -21650.613,E2 -21650.613} C_VEL
LIN {X 0,Y 217.675,Z 519.365,A -85,B 0,C 180,E1 -21652.421,E2 -21652.421} C_VEL
LIN {X 0,Y 218.784,Z 538.806,A -85,B 0,C 180,E1 -21653.425,E2 -21653.425} C_VEL
LIN {X 0,Y 215.755,Z 601.979,A -85,B 0,C 180,E1 -21655.388,E2 -21655.388} C_VEL
LIN {X 0,Y 214.489,Z 615.693,A -85,B 0,C 180,E1 -21656.078,E2 -21656.078} C_VEL
LIN {X 0,Y 212.705,Z 627.27,A -85,B 0,C 180,E1 -21656.963,E2 -21656.963} C_VEL
LIN {X 0,Y 210.439,Z 639.231,A -85,B 0,C 180,E1 -21658.264,E2 -21658.264} C_VEL
LIN {X 0,Y 207.591,Z 651.455,A -85,B 0,C 180,E1 -21660.042,E2 -21660.042} C_VEL
LIN {X 0,Y 204.539,Z 662.169,A -85,B 0,C 180,E1 -21662.085,E2 -21662.085} C_VEL
LIN {X 0,Y 201.281,Z 672.67,A -85,B 0,C 180,E1 -21664.676,E2 -21664.676} C_VEL
LIN {X 0,Y 198.36,Z 681.731,A -85,B 0,C 180,E1 -21667.612,E2 -21667.612} C_VEL
LIN {X 0,Y 195.778,Z 689.012,A -85,B 0,C 180,E1 -21670.606,E2 -21670.606} C_VEL
LIN {X 0,Y 193.3,Z 695.672,A -85,B 0,C 180,E1 -21674.175,E2 -21674.175} C_VEL
LIN {X 0,Y 191.888,Z 700.045,A -85,B 0,C 180,E1 -21677.305,E2 -21677.305} C_VEL
LIN {X 0,Y 191.211,Z 702.347,A -85,B 0,C 180,E1 -21679.41,E2 -21679.41} C_VEL
LIN {X 0,Y 190.689,Z 704.222,A -85,B 0,C 180,E1 -21681.522,E2 -21681.522} C_VEL
LIN {X 0,Y 190.381,Z 705.633,A -85,B 0,C 180,E1 -21683.641,E2 -21683.641} C_VEL
LIN {X 0,Y 190.225,Z 706.711,A -85,B 0,C 180,E1 -21685.976,E2 -21685.976} C_VEL
LIN {X 0,Y 190.231,Z 707.453,A -85,B 0,C 180,E1 -21690,E2 -21690} C_VEL
LIN {X 0,Y 190.211,Z 707.227,A -85,B 0,C 180,E1 -21692.117,E2 -21692.117} C_VEL
LIN {X 0,Y 190.24,Z 706.61,A -85,B 0,C 180,E1 -21694.237,E2 -21694.237} C_VEL
LIN {X 0,Y 190.381,Z 705.605,A -85,B 0,C 180,E1 -21696.358,E2 -21696.358} C_VEL
LIN {X 0,Y 190.692,Z 704.176,A -85,B 0,C 180,E1 -21698.477,E2 -21698.477} C_VEL
LIN {X 0,Y 191.527,Z 701.213,A -85,B 0,C 180,E1 -21701.643,E2 -21701.643} C_VEL
LIN {X 0,Y 192.778,Z 697.189,A -85,B 0,C 180,E1 -21704.785,E2 -21704.785} C_VEL
LIN {X 0,Y 194.997,Z 690.988,A -85,B 0,C 180,E1 -21708.383,E2 -21708.383} C_VEL
LIN {X 0,Y 197.385,Z 684.221,A -85,B 0,C 180,E1 -21711.405,E2 -21711.405} C_VEL
LIN {X 0,Y 200.18,Z 675.962,A -85,B 0,C 180,E1 -21714.287,E2 -21714.287} C_VEL
LIN {X 0,Y 203.001,Z 667.006,A -85,B 0,C 180,E1 -21716.748,E2 -21716.748} C_VEL
LIN {X 0,Y 206.192,Z 656.262,A -85,B 0,C 180,E1 -21719.059,E2 -21719.059} C_VEL
LIN {X 0,Y 209.339,Z 644.22,A -85,B 0,C 180,E1 -21721.076,E2 -21721.076} C_VEL
LIN {X 0,Y 215.298,Z 638.604,A -85,B 0,C 180,E1 -21723.706,E2 -21723.706} C_VEL
LIN {X 0,Y 222.675,Z 631.36,A -85,B 0,C 180,E1 -21726.283,E2 -21726.283} C_VEL
LIN {X 0,Y 230.883,Z 622.621,A -85,B 0,C 180,E1 -21728.61,E2 -21728.61} C_VEL
LIN {X 0,Y 238.456,Z 613.715,A -85,B 0,C 180,E1 -21730.421,E2 -21730.421} C_VEL
LIN {X 0,Y 247.595,Z 601.655,A -85,B 0,C 180,E1 -21732.269,E2 -21732.269} C_VEL
LIN {X 0,Y 255.06,Z 590.546,A -85,B 0,C 180,E1 -21733.54,E2 -21733.54} C_VEL
LIN {X 0,Y 263.297,Z 576.381,A -85,B 0,C 180,E1 -21734.75,E2 -21734.75} C_VEL
LIN {X 0,Y 270.26,Z 562.149,A -85,B 0,C 180,E1 -21735.655,E2 -21735.655} C_VEL
LIN {X 0,Y 275.939,Z 548.057,A -85,B 0,C 180,E1 -21736.416,E2 -21736.416} C_VEL
LIN {X 0,Y 276.486,Z 546.476,A -85,B 0,C 180,E1 -21736.661,E2 -21736.661} C_VEL
LIN {X 0,Y 270.89,Z 559.664,A -85,B 0,C 180,E1 -21737.832,E2 -21737.832} C_VEL
LIN {X 0,Y 264.817,Z 571.223,A -85,B 0,C 180,E1 -21739.192,E2 -21739.192} C_VEL
LIN {X 0,Y 258.217,Z 581.729,A -85,B 0,C 180,E1 -21740.742,E2 -21740.742} C_VEL
LIN {X 0,Y 250.71,Z 591.715,A -85,B 0,C 180,E1 -21742.638,E2 -21742.638} C_VEL
LIN {X 0,Y 243.345,Z 599.986,A -85,B 0,C 180,E1 -21744.717,E2 -21744.717} C_VEL
LIN {X 0,Y 236.996,Z 606.075,A -85,B 0,C 180,E1 -21746.728,E2 -21746.728} C_VEL
LIN {X 0,Y 230.945,Z 611.027,A -85,B 0,C 180,E1 -21748.846,E2 -21748.846} C_VEL
LIN {X 0,Y 225.24,Z 614.933,A -85,B 0,C 180,E1 -21751.077,E2 -21751.077} C_VEL
LIN {X 0,Y 219.871,Z 617.911,A -85,B 0,C 180,E1 -21753.417,E2 -21753.417} C_VEL
LIN {X 0,Y 216.526,Z 619.366,A -85,B 0,C 180,E1 -21755.042,E2 -21755.042} C_VEL
LIN {X 0,Y 210.413,Z 621.053,A -85,B 0,C 180,E1 -21758.444,E2 -21758.444} C_VEL
LIN {X 0,Y 205.123,Z 621.205,A -85,B 0,C 180,E1 -21762.04,E2 -21762.04} C_VEL
LIN {X 0,Y 202.81,Z 620.709,A -85,B 0,C 180,E1 -21763.905,E2 -21763.905} C_VEL
LIN {X 0,Y 198.851,Z 618.501,A -85,B 0,C 180,E1 -21767.757,E2 -21767.757} C_VEL
LIN {X 0,Y 196.614,Z 615.813,A -85,B 0,C 180,E1 -21770.744,E2 -21770.744} C_VEL
LIN {X 0,Y 195.003,Z 612.204,A -85,B 0,C 180,E1 -21773.793,E2 -21773.793} C_VEL
LIN {X 0,Y 193.608,Z 607.582,A -85,B 0,C 180,E1 -21776.879,E2 -21776.879} C_VEL
LIN {X 0,Y 192.628,Z 600.798,A -85,B 0,C 180,E1 -21780.523,E2 -21780.523} C_VEL
LIN {X 0,Y 192.391,Z 593.621,A -85,B 0,C 180,E1 -21783.665,E2 -21783.665} C_VEL
LIN {X 0,Y 192.552,Z 584.871,A -85,B 0,C 180,E1 -21786.813,E2 -21786.813} C_VEL
LIN {X 0,Y 193.016,Z 576.168,A -85,B 0,C 180,E1 -21789.431,E2 -21789.431} C_VEL
LIN {X 0,Y 193.656,Z 565.811,A -85,B 0,C 180,E1 -21792.044,E2 -21792.044} C_VEL
LIN {X 0,Y 194.344,Z 554.498,A -85,B 0,C 180,E1 -21794.396,E2 -21794.396} C_VEL
LIN {X 0,Y 195.116,Z 542.051,A -85,B 0,C 180,E1 -21796.479,E2 -21796.479} C_VEL
LIN {X 0,Y 195.996,Z 528.392,A -85,B 0,C 180,E1 -21798.286,E2 -21798.286} C_VEL
LIN {X 0,Y 196.635,Z 514.973,A -85,B 0,C 180,E1 -21799.645,E2 -21799.645} C_VEL
LIN {X 0,Y 197.132,Z 497.545,A -85,B 0,C 180,E1 -21800.886,E2 -21800.886} C_VEL
LIN {X 0,Y 198.68,Z 447.597,A -85,B 0,C 180,E1 -21804.049,E2 -21804.049} C_VEL
LIN {X 0,Y 194.551,Z 432.243,A -85,B 0,C 180,E1 -21805.201,E2 -21805.201} C_VEL
LIN {X 0,Y 194.449,Z 431.064,A -85,B 0,C 180,E1 -21805.627,E2 -21805.627} C_VEL
LIN {X 0,Y 195.18,Z 430.887,A -85,B 0,C 180,E1 -21806.174,E2 -21806.174} C_VEL
LIN {X 0,Y 195.785,Z 431.252,A -85,B 0,C 180,E1 -21806.661,E2 -21806.661} C_VEL
LIN {X 0,Y 196.674,Z 432.666,A -85,B 0,C 180,E1 -21807.681,E2 -21807.681} C_VEL
LIN {X 0,Y 200.789,Z 441.623,A -85,B 0,C 180,E1 -21812.855,E2 -21812.855} C_VEL
LIN {X 0,Y 204.393,Z 450.398,A -85,B 0,C 180,E1 -21817.093,E2 -21817.093} C_VEL
LIN {X 0,Y 207.357,Z 458.935,A -85,B 0,C 180,E1 -21820.681,E2 -21820.681} C_VEL
LIN {X 0,Y 210.01,Z 467.714,A -85,B 0,C 180,E1 -21823.98,E2 -21823.98} C_VEL
LIN {X 0,Y 212.507,Z 477.709,A -85,B 0,C 180,E1 -21827.29,E2 -21827.29} C_VEL
LIN {X 0,Y 214.336,Z 487.299,A -85,B 0,C 180,E1 -21830.193,E2 -21830.193} C_VEL
LIN {X 0,Y 214.289,Z 488.93,A -85,B 0,C 180,E1 -21830.418,E2 -21830.418} C_VEL
LIN {X 0,Y 217.578,Z 515.512,A -85,B 0,C 180,E1 -21832.228,E2 -21832.228} C_VEL
LIN {X 0,Y 219.328,Z 533.387,A -85,B 0,C 180,E1 -21833.301,E2 -21833.301} C_VEL
LIN {X 0,Y 215.948,Z 602.483,A -85,B 0,C 180,E1 -21835.495,E2 -21835.495} C_VEL
LIN {X 0,Y 214.448,Z 615.292,A -85,B 0,C 180,E1 -21836.213,E2 -21836.213} C_VEL
LIN {X 0,Y 212.442,Z 628.241,A -85,B 0,C 180,E1 -21837.34,E2 -21837.34} C_VEL
LIN {X 0,Y 210.051,Z 640.086,A -85,B 0,C 180,E1 -21838.761,E2 -21838.761} C_VEL
LIN {X 0,Y 207.248,Z 651.341,A -85,B 0,C 180,E1 -21840.547,E2 -21840.547} C_VEL
LIN {X 0,Y 204.334,Z 661.507,A -85,B 0,C 180,E1 -21842.611,E2 -21842.611} C_VEL
LIN {X 0,Y 201.794,Z 669.841,A -85,B 0,C 180,E1 -21844.746,E2 -21844.746} C_VEL
LIN {X 0,Y 198.749,Z 678.872,A -85,B 0,C 180,E1 -21847.658,E2 -21847.658} C_VEL
LIN {X 0,Y 196.167,Z 686.116,A -85,B 0,C 180,E1 -21850.647,E2 -21850.647} C_VEL
LIN {X 0,Y 193.705,Z 692.757,A -85,B 0,C 180,E1 -21854.21,E2 -21854.21} C_VEL
LIN {X 0,Y 192.161,Z 697.118,A -85,B 0,C 180,E1 -21857.324,E2 -21857.324} C_VEL
LIN {X 0,Y 191.437,Z 699.412,A -85,B 0,C 180,E1 -21859.423,E2 -21859.423} C_VEL
LIN {X 0,Y 190.858,Z 701.283,A -85,B 0,C 180,E1 -21861.53,E2 -21861.53} C_VEL
LIN {X 0,Y 190.462,Z 702.708,A -85,B 0,C 180,E1 -21863.645,E2 -21863.645} C_VEL
LIN {X 0,Y 190.224,Z 703.79,A -85,B 0,C 180,E1 -21865.987,E2 -21865.987} C_VEL
LIN {X 0,Y 190.16,Z 704.553,A -85,B 0,C 180,E1 -21870,E2 -21870} C_VEL
LIN {X 0,Y 190.224,Z 703.844,A -85,B 0,C 180,E1 -21874.014,E2 -21874.014} C_VEL
LIN {X 0,Y 190.432,Z 702.783,A -85,B 0,C 180,E1 -21876.357,E2 -21876.357} C_VEL
LIN {X 0,Y 190.781,Z 701.401,A -85,B 0,C 180,E1 -21878.474,E2 -21878.474} C_VEL
LIN {X 0,Y 191.727,Z 698.501,A -85,B 0,C 180,E1 -21881.631,E2 -21881.631} C_VEL
LIN {X 0,Y 193.078,Z 694.56,A -85,B 0,C 180,E1 -21884.762,E2 -21884.762} C_VEL
LIN {X 0,Y 194.912,Z 689.453,A -85,B 0,C 180,E1 -21887.848,E2 -21887.848} C_VEL
LIN {X 0,Y 197.366,Z 683.015,A -85,B 0,C 180,E1 -21890.861,E2 -21890.861} C_VEL
LIN {X 0,Y 199.81,Z 676.08,A -85,B 0,C 180,E1 -21893.458,E2 -21893.458} C_VEL
LIN {X 0,Y 202.752,Z 666.837,A -85,B 0,C 180,E1 -21896.229,E2 -21896.229} C_VEL
LIN {X 0,Y 205.477,Z 657.891,A -85,B 0,C 180,E1 -21898.332,E2 -21898.332} C_VEL
LIN {X 0,Y 208.548,Z 646.792,A -85,B 0,C 180,E1 -21900.365,E2 -21900.365} C_VEL
LIN {X 0,Y 211.044,Z 635.959,A -85,B 0,C 180,E1 -21901.915,E2 -21901.915} C_VEL
LIN {X 0,Y 213.267,Z 623.964,A -85,B 0,C 180,E1 -21903.221,E2 -21903.221} C_VEL
LIN {X 0,Y 215.114,Z 611.463,A -85,B 0,C 180,E1 -21904.162,E2 -21904.162} C_VEL
LIN {X 0,Y 216.292,Z 598.705,A -85,B 0,C 180,E1 -21904.797,E2 -21904.797} C_VEL
LIN {X 0,Y 219.389,Z 532.375,A -85,B 0,C 180,E1 -21906.883,E2 -21906.883} C_VEL
LIN {X 0,Y 216.327,Z 503.67,A -85,B 0,C 180,E1 -21908.68,E2 -21908.68} C_VEL
LIN {X 0,Y 214.301,Z 487.881,A -85,B 0,C 180,E1 -21909.835,E2 -21909.835} C_VEL
LIN {X 0,Y 213.807,Z 484.02,A -85,B 0,C 180,E1 -21910.884,E2 -21910.884} C_VEL
LIN {X 0,Y 211.548,Z 473.442,A -85,B 0,C 180,E1 -21914.24,E2 -21914.24} C_VEL
LIN {X 0,Y 208.815,Z 463.487,A -85,B 0,C 180,E1 -21917.77,E2 -21917.77} C_VEL
LIN {X 0,Y 206.283,Z 455.506,A -85,B 0,C 180,E1 -21920.93,E2 -21920.93} C_VEL
LIN {X 0,Y 203.147,Z 447.219,A -85,B 0,C 180,E1 -21924.586,E2 -21924.586} C_VEL
LIN {X 0,Y 200.15,Z 439.982,A -85,B 0,C 180,E1 -21928.217,E2 -21928.217} C_VEL
LIN {X 0,Y 196.861,Z 432.974,A -85,B 0,C 180,E1 -21932.348,E2 -21932.348} C_VEL
LIN {X 0,Y 194.429,Z 428.368,A -85,B 0,C 180,E1 -21935.519,E2 -21935.519} C_VEL
LIN {X 0,Y 192.646,Z 424.767,A -85,B 0,C 180,E1 -21938.323,E2 -21938.323} C_VEL
LIN {X 0,Y 192.697,Z 424.454,A -85,B 0,C 180,E1 -21941.492,E2 -21941.492} C_VEL
LIN {X 0,Y 192.723,Z 424.48,A -85,B 0,C 180,E1 -21945.21,E2 -21945.21} C_VEL
LIN {X 0,Y 192.948,Z 424.419,A -85,B 0,C 180,E1 -21949.567,E2 -21949.567} C_VEL
LIN {X 0,Y 192.968,Z 424.421,A -85,B 0,C 180,E1 -21953.727,E2 -21953.727} C_VEL
LIN {X 0,Y 193.232,Z 424.4,A -85,B 0,C 180,E1 -21957.916,E2 -21957.916} C_VEL
LIN {X 0,Y 193.416,Z 424.377,A -85,B 0,C 180,E1 -21960,E2 -21960} C_VEL
LIN {X 0,Y 192.934,Z 424.423,A -85,B 0,C 180,E1 -21964.178,E2 -21964.178} C_VEL
LIN {X 0,Y 193.024,Z 424.41,A -85,B 0,C 180,E1 -21968.374,E2 -21968.374} C_VEL
LIN {X 0,Y 192.777,Z 424.466,A -85,B 0,C 180,E1 -21972.635,E2 -21972.635} C_VEL
LIN {X 0,Y 192.697,Z 424.46,A -85,B 0,C 180,E1 -21978.508,E2 -21978.508} C_VEL
LIN {X 0,Y 192.613,Z 424.465,A -85,B 0,C 180,E1 -21984.188,E2 -21984.188} C_VEL
LIN {X 0,Y 192.656,Z 424.625,A -85,B 0,C 180,E1 -21988.309,E2 -21988.309} C_VEL
LIN {X 0,Y 192.828,Z 425.625,A -85,B 0,C 180,E1 -21989.134,E2 -21989.134} C_VEL
LIN {X 0,Y 193.877,Z 427.782,A -85,B 0,C 180,E1 -21990.497,E2 -21990.497} C_VEL
LIN {X 0,Y 195.001,Z 428.985,A -85,B 0,C 180,E1 -21991.506,E2 -21991.506} C_VEL
LIN {X 0,Y 198.9,Z 435.581,A -85,B 0,C 180,E1 -21995.257,E2 -21995.257} C_VEL
LIN {X 0,Y 202.987,Z 442.392,A -85,B 0,C 180,E1 -21998.551,E2 -21998.551} C_VEL
LIN {X 0,Y 205.204,Z 446.47,A -85,B 0,C 180,E1 -22000.246,E2 -22000.246} C_VEL
LIN {X 0,Y 206.68,Z 450.049,A -85,B 0,C 180,E1 -22001.487,E2 -22001.487} C_VEL
LIN {X 0,Y 207.532,Z 454.325,A -85,B 0,C 180,E1 -22002.602,E2 -22002.602} C_VEL
LIN {X 0,Y 208.902,Z 470.305,A -85,B 0,C 180,E1 -22005.965,E2 -22005.965} C_VEL
LIN {X 0,Y 210.414,Z 480.139,A -85,B 0,C 180,E1 -22008.085,E2 -22008.085} C_VEL
LIN {X 0,Y 209.474,Z 488.846,A -85,B 0,C 180,E1 -22009.329,E2 -22009.329} C_VEL
LIN {X 0,Y 212.075,Z 520.15,A -85,B 0,C 180,E1 -22011.277,E2 -22011.277} C_VEL
LIN {X 0,Y 213.103,Z 539.502,A -85,B 0,C 180,E1 -22012.309,E2 -22012.309} C_VEL
LIN {X 0,Y 209.969,Z 602.025,A -85,B 0,C 180,E1 -22014.291,E2 -22014.291} C_VEL
LIN {X 0,Y 208.649,Z 615.695,A -85,B 0,C 180,E1 -22014.993,E2 -22014.993} C_VEL
LIN {X 0,Y 206.791,Z 627.249,A -85,B 0,C 180,E1 -22015.89,E2 -22015.89} C_VEL
LIN {X 0,Y 204.431,Z 639.201,A -85,B 0,C 180,E1 -22017.216,E2 -22017.216} C_VEL
LIN {X 0,Y 201.478,Z 651.417,A -85,B 0,C 180,E1 -22019.035,E2 -22019.035} C_VEL
LIN {X 0,Y 198.288,Z 662.127,A -85,B 0,C 180,E1 -22021.123,E2 -22021.123} C_VEL
LIN {X 0,Y 194.861,Z 672.624,A -85,B 0,C 180,E1 -22023.78,E2 -22023.78} C_VEL
LIN {X 0,Y 191.804,Z 681.682,A -85,B 0,C 180,E1 -22026.802,E2 -22026.802} C_VEL
LIN {X 0,Y 189.092,Z 688.962,A -85,B 0,C 180,E1 -22029.891,E2 -22029.891} C_VEL
LIN {X 0,Y 186.464,Z 695.621,A -85,B 0,C 180,E1 -22033.579,E2 -22033.579} C_VEL
LIN {X 0,Y 184.936,Z 699.992,A -85,B 0,C 180,E1 -22036.819,E2 -22036.819} C_VEL
LIN {X 0,Y 184.205,Z 702.294,A -85,B 0,C 180,E1 -22039.002,E2 -22039.002} C_VEL
LIN {X 0,Y 183.658,Z 704.169,A -85,B 0,C 180,E1 -22041.195,E2 -22041.195} C_VEL
LIN {X 0,Y 183.316,Z 705.58,A -85,B 0,C 180,E1 -22043.395,E2 -22043.395} C_VEL
LIN {X 0,Y 183.13,Z 706.796,A -85,B 0,C 180,E1 -22046.203,E2 -22046.203} C_VEL
LIN {X 0,Y 183.139,Z 707.399,A -85,B 0,C 180,E1 -22050,E2 -22050} C_VEL
LIN {X 0,Y 183.11,Z 706.809,A -85,B 0,C 180,E1 -22053.702,E2 -22053.702} C_VEL
LIN {X 0,Y 183.317,Z 705.55,A -85,B 0,C 180,E1 -22056.604,E2 -22056.604} C_VEL
LIN {X 0,Y 183.66,Z 704.122,A -85,B 0,C 180,E1 -22058.804,E2 -22058.804} C_VEL
LIN {X 0,Y 184.542,Z 701.158,A -85,B 0,C 180,E1 -22062.09,E2 -22062.09} C_VEL
LIN {X 0,Y 185.881,Z 697.135,A -85,B 0,C 180,E1 -22065.347,E2 -22065.347} C_VEL
LIN {X 0,Y 188.251,Z 690.934,A -85,B 0,C 180,E1 -22069.066,E2 -22069.066} C_VEL
LIN {X 0,Y 190.782,Z 684.168,A -85,B 0,C 180,E1 -22072.184,E2 -22072.184} C_VEL
LIN {X 0,Y 193.278,Z 677.189,A -85,B 0,C 180,E1 -22074.74,E2 -22074.74} C_VEL
LIN {X 0,Y 196.039,Z 668.879,A -85,B 0,C 180,E1 -22077.199,E2 -22077.199} C_VEL
LIN {X 0,Y 199.319,Z 658.534,A -85,B 0,C 180,E1 -22079.58,E2 -22079.58} C_VEL
LIN {X 0,Y 202.542,Z 646.886,A -85,B 0,C 180,E1 -22081.656,E2 -22081.656} C_VEL
LIN {X 0,Y 203.293,Z 644.435,A -85,B 0,C 180,E1 -22082.108,E2 -22082.108} C_VEL
LIN {X 0,Y 209.453,Z 639.347,A -85,B 0,C 180,E1 -22084.779,E2 -22084.779} C_VEL
LIN {X 0,Y 218.198,Z 631.652,A -85,B 0,C 180,E1 -22087.733,E2 -22087.733} C_VEL
LIN {X 0,Y 226.713,Z 623.421,A -85,B 0,C 180,E1 -22090.034,E2 -22090.034} C_VEL
LIN {X 0,Y 235.88,Z 613.472,A -85,B 0,C 180,E1 -22092.097,E2 -22092.097} C_VEL
LIN {X 0,Y 244.249,Z 603.328,A -85,B 0,C 180,E1 -22093.676,E2 -22093.676} C_VEL
LIN {X 0,Y 252.337,Z 592.305,A -85,B 0,C 180,E1 -22094.97,E2 -22094.97} C_VEL
LIN {X 0,Y 261.598,Z 577.698,A -85,B 0,C 180,E1 -22096.221,E2 -22096.221} C_VEL
LIN {X 0,Y 266.484,Z 568.765,A -85,B 0,C 180,E1 -22096.814,E2 -22096.814} C_VEL
LIN {X 0,Y 266.282,Z 568.944,A -85,B 0,C 180,E1 -22097.186,E2 -22097.186} C_VEL
LIN {X 0,Y 259.974,Z 579.076,A -85,B 0,C 180,E1 -22098.523,E2 -22098.523} C_VEL
LIN {X 0,Y 252.507,Z 589.151,A -85,B 0,C 180,E1 -22100.196,E2 -22100.196} C_VEL
LIN {X 0,Y 245.271,Z 597.474,A -85,B 0,C 180,E1 -22101.971,E2 -22101.971} C_VEL
LIN {X 0,Y 238.315,Z 604.282,A -85,B 0,C 180,E1 -22103.857,E2 -22103.857} C_VEL
LIN {X 0,Y 231.721,Z 609.818,A -85,B 0,C 180,E1 -22105.868,E2 -22105.868} C_VEL
LIN {X 0,Y 223.427,Z 615.571,A -85,B 0,C 180,E1 -22108.734,E2 -22108.734} C_VEL
LIN {X 0,Y 217.579,Z 618.743,A -85,B 0,C 180,E1 -22111.019,E2 -22111.019} C_VEL
LIN {X 0,Y 210.41,Z 621.53,A -85,B 0,C 180,E1 -22114.264,E2 -22114.264} C_VEL
LIN {X 0,Y 204.016,Z 622.785,A -85,B 0,C 180,E1 -22117.733,E2 -22117.733} C_VEL
LIN {X 0,Y 198.499,Z 622.473,A -85,B 0,C 180,E1 -22121.419,E2 -22121.419} C_VEL
LIN {X 0,Y 193.911,Z 620.643,A -85,B 0,C 180,E1 -22125.303,E2 -22125.303} C_VEL
LIN {X 0,Y 191.953,Z 619.157,A -85,B 0,C 180,E1 -22127.31,E2 -22127.31} C_VEL
LIN {X 0,Y 189.634,Z 616.14,A -85,B 0,C 180,E1 -22130.4,E2 -22130.4} C_VEL
LIN {X 0,Y 187.953,Z 612.209,A -85,B 0,C 180,E1 -22133.559,E2 -22133.559} C_VEL
LIN {X 0,Y 186.512,Z 607.268,A -85,B 0,C 180,E1 -22136.76,E2 -22136.76} C_VEL
LIN {X 0,Y 185.546,Z 600.032,A -85,B 0,C 180,E1 -22140.543,E2 -22140.543} C_VEL
LIN {X 0,Y 185.346,Z 592.45,A -85,B 0,C 180,E1 -22143.805,E2 -22143.805} C_VEL
LIN {X 0,Y 185.548,Z 583.31,A -85,B 0,C 180,E1 -22147.071,E2 -22147.071} C_VEL
LIN {X 0,Y 186.11,Z 573.06,A -85,B 0,C 180,E1 -22150.057,E2 -22150.057} C_VEL
LIN {X 0,Y 186.77,Z 561.9,A -85,B 0,C 180,E1 -22152.744,E2 -22152.744} C_VEL
LIN {X 0,Y 187.619,Z 549.354,A -85,B 0,C 180,E1 -22155.202,E2 -22155.202} C_VEL
LIN {X 0,Y 188.462,Z 535.546,A -85,B 0,C 180,E1 -22157.358,E2 -22157.358} C_VEL
LIN {X 0,Y 189.345,Z 521.001,A -85,B 0,C 180,E1 -22159.093,E2 -22159.093} C_VEL
LIN {X 0,Y 189.789,Z 505.691,A -85,B 0,C 180,E1 -22160.385,E2 -22160.385} C_VEL
LIN {X 0,Y 191.615,Z 448.704,A -85,B 0,C 180,E1 -22164.156,E2 -22164.156} C_VEL
LIN {X 0,Y 188.897,Z 438.809,A -85,B 0,C 180,E1 -22164.985,E2 -22164.985} C_VEL
LIN {X 0,Y 188.85,Z 437.671,A -85,B 0,C 180,E1 -22165.453,E2 -22165.453} C_VEL
LIN {X 0,Y 190.343,Z 437.33,A -85,B 0,C 180,E1 -22166.3,E2 -22166.3} C_VEL
LIN {X 0,Y 191.846,Z 437.68,A -85,B 0,C 180,E1 -22167.253,E2 -22167.253} C_VEL
LIN {X 0,Y 194.993,Z 444.759,A -85,B 0,C 180,E1 -22171.508,E2 -22171.508} C_VEL
LIN {X 0,Y 197.942,Z 451.861,A -85,B 0,C 180,E1 -22175.252,E2 -22175.252} C_VEL
LIN {X 0,Y 200.922,Z 460.228,A -85,B 0,C 180,E1 -22179.022,E2 -22179.022} C_VEL
LIN {X 0,Y 203.954,Z 470.147,A -85,B 0,C 180,E1 -22182.967,E2 -22182.967} C_VEL
LIN {X 0,Y 206.51,Z 480.374,A -85,B 0,C 180,E1 -22186.476,E2 -22186.476} C_VEL
LIN {X 0,Y 208.079,Z 488.384,A -85,B 0,C 180,E1 -22188.958,E2 -22188.958} C_VEL
LIN {X 0,Y 208.909,Z 490.887,A -85,B 0,C 180,E1 -22189.278,E2 -22189.278} C_VEL
LIN {X 0,Y 212.016,Z 516.889,A -85,B 0,C 180,E1 -22191.115,E2 -22191.115} C_VEL
LIN {X 0,Y 213.599,Z 534.882,A -85,B 0,C 180,E1 -22192.211,E2 -22192.211} C_VEL
LIN {X 0,Y 210.147,Z 602.479,A -85,B 0,C 180,E1 -22194.4,E2 -22194.4} C_VEL
LIN {X 0,Y 208.593,Z 615.318,A -85,B 0,C 180,E1 -22195.13,E2 -22195.13} C_VEL
LIN {X 0,Y 206.514,Z 628.278,A -85,B 0,C 180,E1 -22196.28,E2 -22196.28} C_VEL
LIN {X 0,Y 204.02,Z 640.129,A -85,B 0,C 180,E1 -22197.728,E2 -22197.728} C_VEL
LIN {X 0,Y 201.099,Z 651.388,A -85,B 0,C 180,E1 -22199.553,E2 -22199.553} C_VEL
LIN {X 0,Y 198.035,Z 661.557,A -85,B 0,C 180,E1 -22201.663,E2 -22201.663} C_VEL
LIN {X 0,Y 195.376,Z 669.893,A -85,B 0,C 180,E1 -22203.855,E2 -22203.855} C_VEL
LIN {X 0,Y 192.69,Z 677.583,A -85,B 0,C 180,E1 -22206.347,E2 -22206.347} C_VEL
LIN {X 0,Y 189.87,Z 685.073,A -85,B 0,C 180,E1 -22209.412,E2 -22209.412} C_VEL
LIN {X 0,Y 187.467,Z 691.082,A -85,B 0,C 180,E1 -22212.548,E2 -22212.548} C_VEL
LIN {X 0,Y 185.731,Z 695.833,A -85,B 0,C 180,E1 -22215.762,E2 -22215.762} C_VEL
LIN {X 0,Y 184.44,Z 699.467,A -85,B 0,C 180,E1 -22219.017,E2 -22219.017} C_VEL
LIN {X 0,Y 183.823,Z 701.337,A -85,B 0,C 180,E1 -22221.204,E2 -22221.204} C_VEL
LIN {X 0,Y 183.402,Z 702.762,A -85,B 0,C 180,E1 -22223.399,E2 -22223.399} C_VEL
LIN {X 0,Y 183.131,Z 703.978,A -85,B 0,C 180,E1 -22226.204,E2 -22226.204} C_VEL
LIN {X 0,Y 183.071,Z 704.607,A -85,B 0,C 180,E1 -22230,E2 -22230} C_VEL
LIN {X 0,Y 183.097,Z 704.088,A -85,B 0,C 180,E1 -22233.634,E2 -22233.634} C_VEL
LIN {X 0,Y 183.378,Z 702.837,A -85,B 0,C 180,E1 -22236.603,E2 -22236.603} C_VEL
LIN {X 0,Y 183.761,Z 701.454,A -85,B 0,C 180,E1 -22238.8,E2 -22238.8} C_VEL
LIN {X 0,Y 184.77,Z 698.553,A -85,B 0,C 180,E1 -22242.076,E2 -22242.076} C_VEL
LIN {X 0,Y 186.204,Z 694.612,A -85,B 0,C 180,E1 -22245.32,E2 -22245.32} C_VEL
LIN {X 0,Y 188.152,Z 689.503,A -85,B 0,C 180,E1 -22248.512,E2 -22248.512} C_VEL
LIN {X 0,Y 190.729,Z 683.065,A -85,B 0,C 180,E1 -22251.622,E2 -22251.622} C_VEL
LIN {X 0,Y 193.788,Z 674.806,A -85,B 0,C 180,E1 -22254.751,E2 -22254.751} C_VEL
LIN {X 0,Y 196.393,Z 666.882,A -85,B 0,C 180,E1 -22257.147,E2 -22257.147} C_VEL
LIN {X 0,Y 199.258,Z 657.932,A -85,B 0,C 180,E1 -22259.3,E2 -22259.3} C_VEL
LIN {X 0,Y 202.452,Z 646.828,A -85,B 0,C 180,E1 -22261.381,E2 -22261.381} C_VEL
LIN {X 0,Y 205.051,Z 635.99,A -85,B 0,C 180,E1 -22262.964,E2 -22262.964} C_VEL
LIN {X 0,Y 207.374,Z 623.982,A -85,B 0,C 180,E1 -22264.294,E2 -22264.294} C_VEL
LIN {X 0,Y 209.292,Z 611.461,A -85,B 0,C 180,E1 -22265.251,E2 -22265.251} C_VEL
LIN {X 0,Y 210.517,Z 598.661,A -85,B 0,C 180,E1 -22265.896,E2 -22265.896} C_VEL
LIN {X 0,Y 213.727,Z 533.189,A -85,B 0,C 180,E1 -22267.993,E2 -22267.993} C_VEL
LIN {X 0,Y 210.689,Z 504.106,A -85,B 0,C 180,E1 -22269.895,E2 -22269.895} C_VEL
LIN {X 0,Y 208.814,Z 490.015,A -85,B 0,C 180,E1 -22270.951,E2 -22270.951} C_VEL
LIN {X 0,Y 208.006,Z 487.853,A -85,B 0,C 180,E1 -22271.3,E2 -22271.3} C_VEL
LIN {X 0,Y 206.093,Z 478.526,A -85,B 0,C 180,E1 -22274.264,E2 -22274.264} C_VEL
LIN {X 0,Y 203.808,Z 469.555,A -85,B 0,C 180,E1 -22277.438,E2 -22277.438} C_VEL
LIN {X 0,Y 200.679,Z 459.258,A -85,B 0,C 180,E1 -22281.632,E2 -22281.632} C_VEL
LIN {X 0,Y 197.694,Z 451.168,A -85,B 0,C 180,E1 -22285.333,E2 -22285.333} C_VEL
LIN {X 0,Y 195.21,Z 444.985,A -85,B 0,C 180,E1 -22288.531,E2 -22288.531} C_VEL
LIN {X 0,Y 192.052,Z 438.007,A -85,B 0,C 180,E1 -22292.778,E2 -22292.778} C_VEL
LIN {X 0,Y 188.897,Z 432.264,A -85,B 0,C 180,E1 -22297.004,E2 -22297.004} C_VEL
LIN {X 0,Y 188.279,Z 430.85,A -85,B 0,C 180,E1 -22298.082,E2 -22298.082} C_VEL
LIN {X 0,Y 185.685,Z 425.593,A -85,B 0,C 180,E1 -22302.942,E2 -22302.942} C_VEL
LIN {X 0,Y 185.708,Z 425.328,A -85,B 0,C 180,E1 -22306.875,E2 -22306.875} C_VEL
LIN {X 0,Y 185.978,Z 425.309,A -85,B 0,C 180,E1 -22311.306,E2 -22311.306} C_VEL
LIN {X 0,Y 186.178,Z 425.275,A -85,B 0,C 180,E1 -22317.837,E2 -22317.837} C_VEL
LIN {X 0,Y 186.382,Z 425.251,A -85,B 0,C 180,E1 -22320,E2 -22320} C_VEL
LIN {X 0,Y 185.882,Z 425.303,A -85,B 0,C 180,E1 -22324.337,E2 -22324.337} C_VEL
LIN {X 0,Y 185.975,Z 425.284,A -85,B 0,C 180,E1 -22328.694,E2 -22328.694} C_VEL
LIN {X 0,Y 185.701,Z 425.354,A -85,B 0,C 180,E1 -22333.125,E2 -22333.125} C_VEL
LIN {X 0,Y 185.627,Z 425.344,A -85,B 0,C 180,E1 -22338.821,E2 -22338.821} C_VEL
LIN {X 0,Y 185.633,Z 425.537,A -85,B 0,C 180,E1 -22343.719,E2 -22343.719} C_VEL
LIN {X 0,Y 185.911,Z 426.938,A -85,B 0,C 180,E1 -22344.867,E2 -22344.867} C_VEL
LIN {X 0,Y 187.248,Z 429.18,A -85,B 0,C 180,E1 -22346.769,E2 -22346.769} C_VEL
LIN {X 0,Y 188.266,Z 430.085,A -85,B 0,C 180,E1 -22347.816,E2 -22347.816} C_VEL
LIN {X 0,Y 189.446,Z 432.647,A -85,B 0,C 180,E1 -22349.497,E2 -22349.497} C_VEL
LIN {X 0,Y 190.948,Z 434.64,A -85,B 0,C 180,E1 -22351.016,E2 -22351.016} C_VEL
LIN {X 0,Y 194.669,Z 440.858,A -85,B 0,C 180,E1 -22354.654,E2 -22354.654} C_VEL
LIN {X 0,Y 198.839,Z 448.101,A -85,B 0,C 180,E1 -22358.21,E2 -22358.21} C_VEL
LIN {X 0,Y 203.646,Z 457.235,A -85,B 0,C 180,E1 -22361.928,E2 -22361.928} C_VEL
LIN {X 0,Y 208.265,Z 466.604,A -85,B 0,C 180,E1 -22365.126,E2 -22365.126} C_VEL
LIN {X 0,Y 208.902,Z 470.305,A -85,B 0,C 180,E1 -22365.965,E2 -22365.965} C_VEL
LIN {X 0,Y 209.068,Z 473.523,A -85,B 0,C 180,E1 -22366.571,E2 -22366.571} C_VEL
LIN {X 0,Y 208.4,Z 478.81,A -85,B 0,C 180,E1 -22367.268,E2 -22367.268} C_VEL
LIN {X 0,Y 207.144,Z 484.347,A -85,B 0,C 180,E1 -22367.769,E2 -22367.769} C_VEL
LIN {X 0,Y 205.149,Z 494.047,A -85,B 0,C 180,E1 -22368.387,E2 -22368.387} C_VEL
LIN {X 0,Y 204.976,Z 499.955,A -85,B 0,C 180,E1 -22368.747,E2 -22368.747} C_VEL
LIN {X 0,Y 207.281,Z 532.878,A -85,B 0,C 180,E1 -22370.763,E2 -22370.763} C_VEL
LIN {X 0,Y 207.476,Z 540.806,A -85,B 0,C 180,E1 -22371.152,E2 -22371.152} C_VEL
LIN {X 0,Y 204.253,Z 602.144,A -85,B 0,C 180,E1 -22373.134,E2 -22373.134} C_VEL
LIN {X 0,Y 202.882,Z 615.699,A -85,B 0,C 180,E1 -22373.844,E2 -22373.844} C_VEL
LIN {X 0,Y 200.946,Z 627.227,A -85,B 0,C 180,E1 -22374.754,E2 -22374.754} C_VEL
LIN {X 0,Y 198.485,Z 639.169,A -85,B 0,C 180,E1 -22376.104,E2 -22376.104} C_VEL
LIN {X 0,Y 195.416,Z 651.38,A -85,B 0,C 180,E1 -22377.962,E2 -22377.962} C_VEL
LIN {X 0,Y 192.111,Z 662.084,A -85,B 0,C 180,E1 -22380.102,E2 -22380.102} C_VEL
LIN {X 0,Y 188.508,Z 672.578,A -85,B 0,C 180,E1 -22382.825,E2 -22382.825} C_VEL
LIN {X 0,Y 185.271,Z 681.634,A -85,B 0,C 180,E1 -22385.934,E2 -22385.934} C_VEL
LIN {X 0,Y 182.433,Z 688.912,A -85,B 0,C 180,E1 -22389.124,E2 -22389.124} C_VEL
LIN {X 0,Y 180.354,Z 693.839,A -85,B 0,C 180,E1 -22391.835,E2 -22391.835} C_VEL
LIN {X 0,Y 178.508,Z 698.604,A -85,B 0,C 180,E1 -22395.172,E2 -22395.172} C_VEL
LIN {X 0,Y 177.219,Z 702.241,A -85,B 0,C 180,E1 -22398.563,E2 -22398.563} C_VEL
LIN {X 0,Y 176.626,Z 704.115,A -85,B 0,C 180,E1 -22400.841,E2 -22400.841} C_VEL
LIN {X 0,Y 176.251,Z 705.526,A -85,B 0,C 180,E1 -22403.129,E2 -22403.129} C_VEL
LIN {X 0,Y 176.016,Z 706.892,A -85,B 0,C 180,E1 -22406.567,E2 -22406.567} C_VEL
LIN {X 0,Y 176.049,Z 707.345,A -85,B 0,C 180,E1 -22410,E2 -22410} C_VEL
LIN {X 0,Y 176.016,Z 706.878,A -85,B 0,C 180,E1 -22413.432,E2 -22413.432} C_VEL
LIN {X 0,Y 176.251,Z 705.496,A -85,B 0,C 180,E1 -22416.87,E2 -22416.87} C_VEL
LIN {X 0,Y 176.628,Z 704.067,A -85,B 0,C 180,E1 -22419.158,E2 -22419.158} C_VEL
LIN {X 0,Y 177.576,Z 701.103,A -85,B 0,C 180,E1 -22422.572,E2 -22422.572} C_VEL
LIN {X 0,Y 179.009,Z 697.08,A -85,B 0,C 180,E1 -22425.951,E2 -22425.951} C_VEL
LIN {X 0,Y 181.545,Z 690.88,A -85,B 0,C 180,E1 -22429.799,E2 -22429.799} C_VEL
LIN {X 0,Y 184.223,Z 684.116,A -85,B 0,C 180,E1 -22433.019,E2 -22433.019} C_VEL
LIN {X 0,Y 186.799,Z 677.195,A -85,B 0,C 180,E1 -22435.636,E2 -22435.636} C_VEL
LIN {X 0,Y 189.745,Z 668.829,A -85,B 0,C 180,E1 -22438.18,E2 -22438.18} C_VEL
LIN {X 0,Y 193.172,Z 658.486,A -85,B 0,C 180,E1 -22440.62,E2 -22440.62} C_VEL
LIN {X 0,Y 196.521,Z 646.841,A -85,B 0,C 180,E1 -22442.745,E2 -22442.745} C_VEL
LIN {X 0,Y 197.206,Z 644.698,A -85,B 0,C 180,E1 -22443.149,E2 -22443.149} C_VEL
LIN {X 0,Y 203.68,Z 639.958,A -85,B 0,C 180,E1 -22445.915,E2 -22445.915} C_VEL
LIN {X 0,Y 212.657,Z 632.937,A -85,B 0,C 180,E1 -22448.897,E2 -22448.897} C_VEL
LIN {X 0,Y 221.387,Z 625.395,A -85,B 0,C 180,E1 -22451.202,E2 -22451.202} C_VEL
LIN {X 0,Y 230.753,Z 616.301,A -85,B 0,C 180,E1 -22453.258,E2 -22453.258} C_VEL
LIN {X 0,Y 240.749,Z 605.377,A -85,B 0,C 180,E1 -22455.065,E2 -22455.065} C_VEL
LIN {X 0,Y 249.015,Z 595.137,A -85,B 0,C 180,E1 -22456.321,E2 -22456.321} C_VEL
LIN {X 0,Y 256.634,Z 584.466,A -85,B 0,C 180,E1 -22457.298,E2 -22457.298} C_VEL
LIN {X 0,Y 255.745,Z 585.526,A -85,B 0,C 180,E1 -22457.68,E2 -22457.68} C_VEL
LIN {X 0,Y 247.986,Z 594.686,A -85,B 0,C 180,E1 -22459.32,E2 -22459.32} C_VEL
LIN {X 0,Y 240.516,Z 602.25,A -85,B 0,C 180,E1 -22461.079,E2 -22461.079} C_VEL
LIN {X 0,Y 233.332,Z 608.438,A -85,B 0,C 180,E1 -22462.958,E2 -22462.958} C_VEL
LIN {X 0,Y 224.265,Z 614.896,A -85,B 0,C 180,E1 -22465.661,E2 -22465.661} C_VEL
LIN {X 0,Y 217.848,Z 618.566,A -85,B 0,C 180,E1 -22467.838,E2 -22467.838} C_VEL
LIN {X 0,Y 211.773,Z 621.314,A -85,B 0,C 180,E1 -22470.146,E2 -22470.146} C_VEL
LIN {X 0,Y 207.943,Z 622.667,A -85,B 0,C 180,E1 -22471.76,E2 -22471.76} C_VEL
LIN {X 0,Y 200.865,Z 624.172,A -85,B 0,C 180,E1 -22475.174,E2 -22475.174} C_VEL
LIN {X 0,Y 194.631,Z 624.199,A -85,B 0,C 180,E1 -22478.833,E2 -22478.833} C_VEL
LIN {X 0,Y 189.352,Z 622.685,A -85,B 0,C 180,E1 -22482.727,E2 -22482.727} C_VEL
LIN {X 0,Y 185.071,Z 619.632,A -85,B 0,C 180,E1 -22486.83,E2 -22486.83} C_VEL
LIN {X 0,Y 182.646,Z 616.309,A -85,B 0,C 180,E1 -22490.029,E2 -22490.029} C_VEL
LIN {X 0,Y 180.89,Z 612.04,A -85,B 0,C 180,E1 -22493.307,E2 -22493.307} C_VEL
LIN {X 0,Y 179.214,Z 605.772,A -85,B 0,C 180,E1 -22497.19,E2 -22497.19} C_VEL
LIN {X 0,Y 178.47,Z 599.135,A -85,B 0,C 180,E1 -22500.564,E2 -22500.564} C_VEL
LIN {X 0,Y 178.298,Z 591.078,A -85,B 0,C 180,E1 -22503.956,E2 -22503.956} C_VEL
LIN {X 0,Y 178.589,Z 581.395,A -85,B 0,C 180,E1 -22507.348,E2 -22507.348} C_VEL
LIN {X 0,Y 179.188,Z 570.818,A -85,B 0,C 180,E1 -22510.416,E2 -22510.416} C_VEL
LIN {X 0,Y 179.928,Z 558.746,A -85,B 0,C 180,E1 -22513.238,E2 -22513.238} C_VEL
LIN {X 0,Y 180.644,Z 546.775,A -85,B 0,C 180,E1 -22515.514,E2 -22515.514} C_VEL
LIN {X 0,Y 181.51,Z 532.997,A -85,B 0,C 180,E1 -22517.608,E2 -22517.608} C_VEL
LIN {X 0,Y 182.353,Z 518.597,A -85,B 0,C 180,E1 -22519.269,E2 -22519.269} C_VEL
LIN {X 0,Y 182.802,Z 503.304,A -85,B 0,C 180,E1 -22520.538,E2 -22520.538} C_VEL
LIN {X 0,Y 184.555,Z 449.803,A -85,B 0,C 180,E1 -22524.27,E2 -22524.27} C_VEL
LIN {X 0,Y 183.387,Z 445.484,A -85,B 0,C 180,E1 -22524.668,E2 -22524.668} C_VEL
LIN {X 0,Y 183.265,Z 444.397,A -85,B 0,C 180,E1 -22525.11,E2 -22525.11} C_VEL
LIN {X 0,Y 184.655,Z 444.025,A -85,B 0,C 180,E1 -22526.019,E2 -22526.019} C_VEL
LIN {X 0,Y 186.706,Z 443.25,A -85,B 0,C 180,E1 -22526.853,E2 -22526.853} C_VEL
LIN {X 0,Y 187.706,Z 444.477,A -85,B 0,C 180,E1 -22527.906,E2 -22527.906} C_VEL
LIN {X 0,Y 190.067,Z 449.747,A -85,B 0,C 180,E1 -22531.176,E2 -22531.176} C_VEL
LIN {X 0,Y 192.922,Z 456.896,A -85,B 0,C 180,E1 -22535.013,E2 -22535.013} C_VEL
LIN {X 0,Y 195.792,Z 465.407,A -85,B 0,C 180,E1 -22538.915,E2 -22538.915} C_VEL
LIN {X 0,Y 198.74,Z 475.388,A -85,B 0,C 180,E1 -22542.901,E2 -22542.901} C_VEL
LIN {X 0,Y 200.926,Z 485.065,A -85,B 0,C 180,E1 -22546.295,E2 -22546.295} C_VEL
LIN {X 0,Y 201.617,Z 488.482,A -85,B 0,C 180,E1 -22547.348,E2 -22547.348} C_VEL
LIN {X 0,Y 203.681,Z 493.205,A -85,B 0,C 180,E1 -22548.109,E2 -22548.109} C_VEL
LIN {X 0,Y 206.553,Z 518.516,A -85,B 0,C 180,E1 -22549.956,E2 -22549.956} C_VEL
LIN {X 0,Y 207.977,Z 535.901,A -85,B 0,C 180,E1 -22551.046,E2 -22551.046} C_VEL
LIN {X 0,Y 204.436,Z 602.474,A -85,B 0,C 180,E1 -22553.246,E2 -22553.246} C_VEL
LIN {X 0,Y 202.817,Z 615.345,A -85,B 0,C 180,E1 -22553.985,E2 -22553.985} C_VEL
LIN {X 0,Y 200.649,Z 628.315,A -85,B 0,C 180,E1 -22555.155,E2 -22555.155} C_VEL
LIN {X 0,Y 198.053,Z 640.173,A -85,B 0,C 180,E1 -22556.631,E2 -22556.631} C_VEL
LIN {X 0,Y 195.017,Z 651.436,A -85,B 0,C 180,E1 -22558.497,E2 -22558.497} C_VEL
LIN {X 0,Y 191.806,Z 661.606,A -85,B 0,C 180,E1 -22560.655,E2 -22560.655} C_VEL
LIN {X 0,Y 189.012,Z 669.944,A -85,B 0,C 180,E1 -22562.904,E2 -22562.904} C_VEL
LIN {X 0,Y 186.209,Z 677.636,A -85,B 0,C 180,E1 -22565.47,E2 -22565.47} C_VEL
LIN {X 0,Y 183.234,Z 685.126,A -85,B 0,C 180,E1 -22568.631,E2 -22568.631} C_VEL
LIN {X 0,Y 180.684,Z 691.136,A -85,B 0,C 180,E1 -22571.87,E2 -22571.87} C_VEL
LIN {X 0,Y 178.846,Z 695.887,A -85,B 0,C 180,E1 -22575.201,E2 -22575.201} C_VEL
LIN {X 0,Y 177.466,Z 699.521,A -85,B 0,C 180,E1 -22578.58,E2 -22578.58} C_VEL
LIN {X 0,Y 176.81,Z 701.392,A -85,B 0,C 180,E1 -22580.852,E2 -22580.852} C_VEL
LIN {X 0,Y 176.345,Z 702.816,A -85,B 0,C 180,E1 -22583.133,E2 -22583.133} C_VEL
LIN {X 0,Y 175.97,Z 704.43,A -85,B 0,C 180,E1 -22587.711,E2 -22587.711} C_VEL
LIN {X 0,Y 175.984,Z 704.661,A -85,B 0,C 180,E1 -22590,E2 -22590} C_VEL
LIN {X 0,Y 175.996,Z 704.249,A -85,B 0,C 180,E1 -22593.32,E2 -22593.32} C_VEL
LIN {X 0,Y 176.325,Z 702.89,A -85,B 0,C 180,E1 -22596.868,E2 -22596.868} C_VEL
LIN {X 0,Y 176.737,Z 701.508,A -85,B 0,C 180,E1 -22599.153,E2 -22599.153} C_VEL
LIN {X 0,Y 177.816,Z 698.606,A -85,B 0,C 180,E1 -22602.556,E2 -22602.556} C_VEL
LIN {X 0,Y 179.333,Z 694.664,A -85,B 0,C 180,E1 -22605.922,E2 -22605.922} C_VEL
LIN {X 0,Y 181.425,Z 689.554,A -85,B 0,C 180,E1 -22609.225,E2 -22609.225} C_VEL
LIN {X 0,Y 184.128,Z 683.114,A -85,B 0,C 180,E1 -22612.439,E2 -22612.439} C_VEL
LIN {X 0,Y 187.143,Z 675.403,A -85,B 0,C 180,E1 -22615.468,E2 -22615.468} C_VEL
LIN {X 0,Y 190.084,Z 666.927,A -85,B 0,C 180,E1 -22618.126,E2 -22618.126} C_VEL
LIN {X 0,Y 193.458,Z 656.833,A -85,B 0,C 180,E1 -22620.571,E2 -22620.571} C_VEL
LIN {X 0,Y 196.799,Z 645.479,A -85,B 0,C 180,E1 -22622.694,E2 -22622.694} C_VEL
LIN {X 0,Y 199.513,Z 634.267,A -85,B 0,C 180,E1 -22624.307,E2 -22624.307} C_VEL
LIN {X 0,Y 201.99,Z 621.526,A -85,B 0,C 180,E1 -22625.648,E2 -22625.648} C_VEL
LIN {X 0,Y 203.875,Z 608.898,A -85,B 0,C 180,E1 -22626.565,E2 -22626.565} C_VEL
LIN {X 0,Y 205.056,Z 595.503,A -85,B 0,C 180,E1 -22627.163,E2 -22627.163} C_VEL
LIN {X 0,Y 208.145,Z 534.01,A -85,B 0,C 180,E1 -22629.163,E2 -22629.163} C_VEL
LIN {X 0,Y 205.242,Z 505.304,A -85,B 0,C 180,E1 -22631.12,E2 -22631.12} C_VEL
LIN {X 0,Y 203.7,Z 493.073,A -85,B 0,C 180,E1 -22632.065,E2 -22632.065} C_VEL
LIN {X 0,Y 201.519,Z 487.957,A -85,B 0,C 180,E1 -22632.914,E2 -22632.914} C_VEL
LIN {X 0,Y 199.447,Z 478.444,A -85,B 0,C 180,E1 -22636.143,E2 -22636.143} C_VEL
LIN {X 0,Y 197.564,Z 471.126,A -85,B 0,C 180,E1 -22638.921,E2 -22638.921} C_VEL
LIN {X 0,Y 195.057,Z 462.884,A -85,B 0,C 180,E1 -22642.437,E2 -22642.437} C_VEL
LIN {X 0,Y 192.303,Z 455.157,A -85,B 0,C 180,E1 -22646.128,E2 -22646.128} C_VEL
LIN {X 0,Y 190.345,Z 450.018,A -85,B 0,C 180,E1 -22648.874,E2 -22648.874} C_VEL
LIN {X 0,Y 187.253,Z 443.041,A -85,B 0,C 180,E1 -22653.231,E2 -22653.231} C_VEL
LIN {X 0,Y 184.276,Z 437.346,A -85,B 0,C 180,E1 -22657.58,E2 -22657.58} C_VEL
LIN {X 0,Y 181.346,Z 431.183,A -85,B 0,C 180,E1 -22663.102,E2 -22663.102} C_VEL
LIN {X 0,Y 179.086,Z 427.847,A -85,B 0,C 180,E1 -22667.535,E2 -22667.535} C_VEL
LIN {X 0,Y 178.854,Z 426.452,A -85,B 0,C 180,E1 -22669.228,E2 -22669.228} C_VEL
LIN {X 0,Y 178.908,Z 426.185,A -85,B 0,C 180,E1 -22670.959,E2 -22670.959} C_VEL
LIN {X 0,Y 179.125,Z 426.151,A -85,B 0,C 180,E1 -22677.751,E2 -22677.751} C_VEL
LIN {X 0,Y 179.347,Z 426.126,A -85,B 0,C 180,E1 -22680,E2 -22680} C_VEL
LIN {X 0,Y 178.831,Z 426.182,A -85,B 0,C 180,E1 -22684.508,E2 -22684.508} C_VEL
LIN {X 0,Y 178.906,Z 426.162,A -85,B 0,C 180,E1 -22689.04,E2 -22689.04} C_VEL
LIN {X 0,Y 178.626,Z 426.226,A -85,B 0,C 180,E1 -22693.655,E2 -22693.655} C_VEL
LIN {X 0,Y 178.627,Z 426.498,A -85,B 0,C 180,E1 -22697.163,E2 -22697.163} C_VEL
LIN {X 0,Y 178.814,Z 427.308,A -85,B 0,C 180,E1 -22698.326,E2 -22698.326} C_VEL
LIN {X 0,Y 179.723,Z 429.46,A -85,B 0,C 180,E1 -22700.606,E2 -22700.606} C_VEL
LIN {X 0,Y 181.252,Z 430.997,A -85,B 0,C 180,E1 -22702.814,E2 -22702.814} C_VEL
LIN {X 0,Y 181.951,Z 432.089,A -85,B 0,C 180,E1 -22703.927,E2 -22703.927} C_VEL
LIN {X 0,Y 183.302,Z 434.822,A -85,B 0,C 180,E1 -22706.163,E2 -22706.163} C_VEL
LIN {X 0,Y 184.253,Z 435.806,A -85,B 0,C 180,E1 -22707.24,E2 -22707.24} C_VEL
LIN {X 0,Y 187.89,Z 442.02,A -85,B 0,C 180,E1 -22711.579,E2 -22711.579} C_VEL
LIN {X 0,Y 191.115,Z 447.444,A -85,B 0,C 180,E1 -22714.75,E2 -22714.75} C_VEL
LIN {X 0,Y 195.907,Z 456.164,A -85,B 0,C 180,E1 -22718.888,E2 -22718.888} C_VEL
LIN {X 0,Y 199.756,Z 463.801,A -85,B 0,C 180,E1 -22721.949,E2 -22721.949} C_VEL
LIN {X 0,Y 203.115,Z 470.933,A -85,B 0,C 180,E1 -22724.439,E2 -22724.439} C_VEL
LIN {X 0,Y 204.671,Z 481.642,A -85,B 0,C 180,E1 -22726.858,E2 -22726.858} C_VEL
LIN {X 0,Y 204.417,Z 485.595,A -85,B 0,C 180,E1 -22727.508,E2 -22727.508} C_VEL
LIN {X 0,Y 204.007,Z 488.954,A -85,B 0,C 180,E1 -22727.998,E2 -22727.998} C_VEL
LIN {X 0,Y 204.976,Z 499.955,A -85,B 0,C 180,E1 -22728.747,E2 -22728.747} C_VEL
LIN {X 0,Y 204.912,Z 505.8,A -85,B 0,C 180,E1 -22728.998,E2 -22728.998} C_VEL
LIN {X 0,Y 201.765,Z 525.431,A -85,B 0,C 180,E1 -22729.126,E2 -22729.126} C_VEL
LIN {X 0,Y 201.661,Z 531.29,A -85,B 0,C 180,E1 -22729.37,E2 -22729.37} C_VEL
LIN {X 0,Y 201.971,Z 541.406,A -85,B 0,C 180,E1 -22729.906,E2 -22729.906} C_VEL
LIN {X 0,Y 198.612,Z 602.509,A -85,B 0,C 180,E1 -22731.922,E2 -22731.922} C_VEL
LIN {X 0,Y 197.18,Z 615.713,A -85,B 0,C 180,E1 -22732.625,E2 -22732.625} C_VEL
LIN {X 0,Y 194.979,Z 628.308,A -85,B 0,C 180,E1 -22733.666,E2 -22733.666} C_VEL
LIN {X 0,Y 192.246,Z 640.871,A -85,B 0,C 180,E1 -22735.165,E2 -22735.165} C_VEL
LIN {X 0,Y 189.436,Z 651.342,A -85,B 0,C 180,E1 -22736.823,E2 -22736.823} C_VEL
LIN {X 0,Y 185.997,Z 662.042,A -85,B 0,C 180,E1 -22739.013,E2 -22739.013} C_VEL
LIN {X 0,Y 182.213,Z 672.532,A -85,B 0,C 180,E1 -22741.804,E2 -22741.804} C_VEL
LIN {X 0,Y 178.772,Z 681.607,A -85,B 0,C 180,E1 -22745.01,E2 -22745.01} C_VEL
LIN {X 0,Y 175.797,Z 688.862,A -85,B 0,C 180,E1 -22748.297,E2 -22748.297} C_VEL
LIN {X 0,Y 173.616,Z 693.788,A -85,B 0,C 180,E1 -22751.104,E2 -22751.104} C_VEL
LIN {X 0,Y 171.61,Z 698.552,A -85,B 0,C 180,E1 -22754.562,E2 -22754.562} C_VEL
LIN {X 0,Y 170.253,Z 702.188,A -85,B 0,C 180,E1 -22758.088,E2 -22758.088} C_VEL
LIN {X 0,Y 169.615,Z 704.062,A -85,B 0,C 180,E1 -22760.459,E2 -22760.459} C_VEL
LIN {X 0,Y 169.182,Z 705.473,A -85,B 0,C 180,E1 -22762.841,E2 -22762.841} C_VEL
LIN {X 0,Y 168.93,Z 706.921,A -85,B 0,C 180,E1 -22766.836,E2 -22766.836} C_VEL
LIN {X 0,Y 168.962,Z 707.291,A -85,B 0,C 180,E1 -22770,E2 -22770} C_VEL
LIN {X 0,Y 168.91,Z 706.932,A -85,B 0,C 180,E1 -22773.038,E2 -22773.038} C_VEL
LIN {X 0,Y 169.182,Z 705.441,A -85,B 0,C 180,E1 -22777.159,E2 -22777.159} C_VEL
LIN {X 0,Y 169.617,Z 704.013,A -85,B 0,C 180,E1 -22779.54,E2 -22779.54} C_VEL
LIN {X 0,Y 170.634,Z 701.049,A -85,B 0,C 180,E1 -22783.093,E2 -22783.093} C_VEL
LIN {X 0,Y 172.164,Z 697.026,A -85,B 0,C 180,E1 -22786.604,E2 -22786.604} C_VEL
LIN {X 0,Y 174.871,Z 690.827,A -85,B 0,C 180,E1 -22790.589,E2 -22790.589} C_VEL
LIN {X 0,Y 177.699,Z 684.087,A -85,B 0,C 180,E1 -22793.903,E2 -22793.903} C_VEL
LIN {X 0,Y 180.406,Z 677.143,A -85,B 0,C 180,E1 -22796.614,E2 -22796.614} C_VEL
LIN {X 0,Y 183.52,Z 668.778,A -85,B 0,C 180,E1 -22799.227,E2 -22799.227} C_VEL
LIN {X 0,Y 187.075,Z 658.438,A -85,B 0,C 180,E1 -22801.732,E2 -22801.732} C_VEL
LIN {X 0,Y 190.592,Z 646.797,A -85,B 0,C 180,E1 -22803.899,E2 -22803.899} C_VEL
LIN {X 0,Y 191.311,Z 644.675,A -85,B 0,C 180,E1 -22804.31,E2 -22804.31} C_VEL
LIN {X 0,Y 197.984,Z 640.425,A -85,B 0,C 180,E1 -22807.118,E2 -22807.118} C_VEL
LIN {X 0,Y 207.214,Z 634.053,A -85,B 0,C 180,E1 -22810.122,E2 -22810.122} C_VEL
LIN {X 0,Y 216.151,Z 627.165,A -85,B 0,C 180,E1 -22812.429,E2 -22812.429} C_VEL
LIN {X 0,Y 225.682,Z 618.898,A -85,B 0,C 180,E1 -22814.481,E2 -22814.481} C_VEL
LIN {X 0,Y 235.87,Z 608.936,A -85,B 0,C 180,E1 -22816.266,E2 -22816.266} C_VEL
LIN {X 0,Y 244.932,Z 598.912,A -85,B 0,C 180,E1 -22817.601,E2 -22817.601} C_VEL
LIN {X 0,Y 245.748,Z 597.82,A -85,B 0,C 180,E1 -22817.941,E2 -22817.941} C_VEL
LIN {X 0,Y 237.051,Z 605.774,A -85,B 0,C 180,E1 -22819.847,E2 -22819.847} C_VEL
LIN {X 0,Y 228.37,Z 612.445,A -85,B 0,C 180,E1 -22822.012,E2 -22822.012} C_VEL
LIN {X 0,Y 218.963,Z 618.215,A -85,B 0,C 180,E1 -22824.708,E2 -22824.708} C_VEL
LIN {X 0,Y 214.473,Z 620.495,A -85,B 0,C 180,E1 -22826.147,E2 -22826.147} C_VEL
LIN {X 0,Y 205.984,Z 623.784,A -85,B 0,C 180,E1 -22829.217,E2 -22829.217} C_VEL
LIN {X 0,Y 198.21,Z 625.58,A -85,B 0,C 180,E1 -22832.552,E2 -22832.552} C_VEL
LIN {X 0,Y 191.268,Z 625.85,A -85,B 0,C 180,E1 -22836.16,E2 -22836.16} C_VEL
LIN {X 0,Y 185.271,Z 624.643,A -85,B 0,C 180,E1 -22840.038,E2 -22840.038} C_VEL
LIN {X 0,Y 180.292,Z 621.937,A -85,B 0,C 180,E1 -22844.165,E2 -22844.165} C_VEL
LIN {X 0,Y 176.373,Z 617.641,A -85,B 0,C 180,E1 -22848.508,E2 -22848.508} C_VEL
LIN {X 0,Y 174.43,Z 613.379,A -85,B 0,C 180,E1 -22851.893,E2 -22851.893} C_VEL
LIN {X 0,Y 172.534,Z 607.09,A -85,B 0,C 180,E1 -22855.912,E2 -22855.912} C_VEL
LIN {X 0,Y 171.459,Z 599.218,A -85,B 0,C 180,E1 -22860,E2 -22860} C_VEL
LIN {X 0,Y 171.247,Z 591.041,A -85,B 0,C 180,E1 -22863.529,E2 -22863.529} C_VEL
LIN {X 0,Y 171.513,Z 581.104,A -85,B 0,C 180,E1 -22867.061,E2 -22867.061} C_VEL
LIN {X 0,Y 172.213,Z 569.316,A -85,B 0,C 180,E1 -22870.483,E2 -22870.483} C_VEL
LIN {X 0,Y 172.869,Z 558.189,A -85,B 0,C 180,E1 -22873.13,E2 -22873.13} C_VEL
LIN {X 0,Y 173.627,Z 545.675,A -85,B 0,C 180,E1 -22875.555,E2 -22875.555} C_VEL
LIN {X 0,Y 174.447,Z 532.353,A -85,B 0,C 180,E1 -22877.587,E2 -22877.587} C_VEL
LIN {X 0,Y 175.281,Z 517.461,A -85,B 0,C 180,E1 -22879.317,E2 -22879.317} C_VEL
LIN {X 0,Y 175.887,Z 496.377,A -85,B 0,C 180,E1 -22881,E2 -22881} C_VEL
LIN {X 0,Y 177.426,Z 452.713,A -85,B 0,C 180,E1 -22884.289,E2 -22884.289} C_VEL
LIN {X 0,Y 177.686,Z 451.177,A -85,B 0,C 180,E1 -22884.699,E2 -22884.699} C_VEL
LIN {X 0,Y 178.799,Z 450.86,A -85,B 0,C 180,E1 -22885.619,E2 -22885.619} C_VEL
LIN {X 0,Y 179.972,Z 450.306,A -85,B 0,C 180,E1 -22886.082,E2 -22886.082} C_VEL
LIN {X 0,Y 182.891,Z 449.561,A -85,B 0,C 180,E1 -22887.46,E2 -22887.46} C_VEL
LIN {X 0,Y 185.219,Z 454.798,A -85,B 0,C 180,E1 -22890.814,E2 -22890.814} C_VEL
LIN {X 0,Y 187.854,Z 461.669,A -85,B 0,C 180,E1 -22894.607,E2 -22894.607} C_VEL
LIN {X 0,Y 190.421,Z 469.777,A -85,B 0,C 180,E1 -22898.451,E2 -22898.451} C_VEL
LIN {X 0,Y 193.353,Z 479.835,A -85,B 0,C 180,E1 -22902.479,E2 -22902.479} C_VEL
LIN {X 0,Y 195.205,Z 488.516,A -85,B 0,C 180,E1 -22905.594,E2 -22905.594} C_VEL
LIN {X 0,Y 198.652,Z 496.418,A -85,B 0,C 180,E1 -22906.953,E2 -22906.953} C_VEL
LIN {X 0,Y 201.334,Z 521.982,A -85,B 0,C 180,E1 -22908.859,E2 -22908.859} C_VEL
LIN {X 0,Y 202.491,Z 535.865,A -85,B 0,C 180,E1 -22909.78,E2 -22909.78} C_VEL
LIN {X 0,Y 198.804,Z 602.47,A -85,B 0,C 180,E1 -22912.024,E2 -22912.024} C_VEL
LIN {X 0,Y 197.127,Z 615.371,A -85,B 0,C 180,E1 -22912.773,E2 -22912.773} C_VEL
LIN {X 0,Y 194.878,Z 628.351,A -85,B 0,C 180,E1 -22913.964,E2 -22913.964} C_VEL
LIN {X 0,Y 192.178,Z 640.216,A -85,B 0,C 180,E1 -22915.47,E2 -22915.47} C_VEL
LIN {X 0,Y 189.008,Z 651.483,A -85,B 0,C 180,E1 -22917.374,E2 -22917.374} C_VEL
LIN {X 0,Y 185.661,Z 661.656,A -85,B 0,C 180,E1 -22919.583,E2 -22919.583} C_VEL
LIN {X 0,Y 182.718,Z 669.995,A -85,B 0,C 180,E1 -22921.889,E2 -22921.889} C_VEL
LIN {X 0,Y 179.189,Z 679.031,A -85,B 0,C 180,E1 -22925.063,E2 -22925.063} C_VEL
LIN {X 0,Y 176.155,Z 686.277,A -85,B 0,C 180,E1 -22928.344,E2 -22928.344} C_VEL
LIN {X 0,Y 173.226,Z 692.92,A -85,B 0,C 180,E1 -22932.285,E2 -22932.285} C_VEL
LIN {X 0,Y 171.425,Z 697.281,A -85,B 0,C 180,E1 -22935.76,E2 -22935.76} C_VEL
LIN {X 0,Y 170.514,Z 699.576,A -85,B 0,C 180,E1 -22938.107,E2 -22938.107} C_VEL
LIN {X 0,Y 169.794,Z 701.446,A -85,B 0,C 180,E1 -22940.47,E2 -22940.47} C_VEL
LIN {X 0,Y 169.287,Z 702.871,A -85,B 0,C 180,E1 -22942.846,E2 -22942.846} C_VEL
LIN {X 0,Y 168.892,Z 704.378,A -85,B 0,C 180,E1 -22947.079,E2 -22947.079} C_VEL
LIN {X 0,Y 168.884,Z 704.715,A -85,B 0,C 180,E1 -22950,E2 -22950} C_VEL
LIN {X 0,Y 168.893,Z 704.409,A -85,B 0,C 180,E1 -22952.922,E2 -22952.922} C_VEL
LIN {X 0,Y 169.269,Z 702.944,A -85,B 0,C 180,E1 -22957.156,E2 -22957.156} C_VEL
LIN {X 0,Y 169.716,Z 701.561,A -85,B 0,C 180,E1 -22959.535,E2 -22959.535} C_VEL
LIN {X 0,Y 170.864,Z 698.659,A -85,B 0,C 180,E1 -22963.075,E2 -22963.075} C_VEL
LIN {X 0,Y 172.482,Z 694.715,A -85,B 0,C 180,E1 -22966.573,E2 -22966.573} C_VEL
LIN {X 0,Y 174.733,Z 689.604,A -85,B 0,C 180,E1 -22969.992,E2 -22969.992} C_VEL
LIN {X 0,Y 177.566,Z 683.163,A -85,B 0,C 180,E1 -22973.316,E2 -22973.316} C_VEL
LIN {X 0,Y 180.52,Z 676.016,A -85,B 0,C 180,E1 -22976.231,E2 -22976.231} C_VEL
LIN {X 0,Y 183.844,Z 666.972,A -85,B 0,C 180,E1 -22979.171,E2 -22979.171} C_VEL
LIN {X 0,Y 187.022,Z 658.015,A -85,B 0,C 180,E1 -22981.427,E2 -22981.427} C_VEL
LIN {X 0,Y 190.461,Z 646.902,A -85,B 0,C 180,E1 -22983.608,E2 -22983.608} C_VEL
LIN {X 0,Y 193.297,Z 636.051,A -85,B 0,C 180,E1 -22985.254,E2 -22985.254} C_VEL
LIN {X 0,Y 195.814,Z 624.016,A -85,B 0,C 180,E1 -22986.634,E2 -22986.634} C_VEL
LIN {X 0,Y 197.999,Z 610.603,A -85,B 0,C 180,E1 -22987.676,E2 -22987.676} C_VEL
LIN {X 0,Y 199.208,Z 598.574,A -85,B 0,C 180,E1 -22988.287,E2 -22988.287} C_VEL
LIN {X 0,Y 202.652,Z 535.066,A -85,B 0,C 180,E1 -22990.388,E2 -22990.388} C_VEL
LIN {X 0,Y 200.005,Z 507.322,A -85,B 0,C 180,E1 -22992.342,E2 -22992.342} C_VEL
LIN {X 0,Y 198.671,Z 496.052,A -85,B 0,C 180,E1 -22993.238,E2 -22993.238} C_VEL
LIN {X 0,Y 195.064,Z 487.842,A -85,B 0,C 180,E1 -22994.729,E2 -22994.729} C_VEL
LIN {X 0,Y 192.803,Z 477.901,A -85,B 0,C 180,E1 -22998.372,E2 -22998.372} C_VEL
LIN {X 0,Y 190.244,Z 468.813,A -85,B 0,C 180,E1 -23002.183,E2 -23002.183} C_VEL
LIN {X 0,Y 187.758,Z 461.264,A -85,B 0,C 180,E1 -23005.842,E2 -23005.842} C_VEL
LIN {X 0,Y 185.506,Z 455.081,A -85,B 0,C 180,E1 -23009.239,E2 -23009.239} C_VEL
LIN {X 0,Y 182.476,Z 448.095,A -85,B 0,C 180,E1 -23013.709,E2 -23013.709} C_VEL
LIN {X 0,Y 179.682,Z 442.456,A -85,B 0,C 180,E1 -23018.187,E2 -23018.187} C_VEL
LIN {X 0,Y 176.827,Z 436.502,A -85,B 0,C 180,E1 -23023.846,E2 -23023.846} C_VEL
LIN {X 0,Y 174.209,Z 431.528,A -85,B 0,C 180,E1 -23030.713,E2 -23030.713} C_VEL
LIN {X 0,Y 172.519,Z 428.076,A -85,B 0,C 180,E1 -23040,E2 -23040} C_VEL
LIN {X 0,Y 172.285,Z 428.046,A -85,B 0,C 180,E1 -23042.338,E2 -23042.338} C_VEL
LIN {X 0,Y 172.547,Z 429.376,A -85,B 0,C 180,E1 -23049.377,E2 -23049.377} C_VEL
LIN {X 0,Y 174.612,Z 432.166,A -85,B 0,C 180,E1 -23056.364,E2 -23056.364} C_VEL
LIN {X 0,Y 178.048,Z 437.707,A -85,B 0,C 180,E1 -23063.249,E2 -23063.249} C_VEL
LIN {X 0,Y 179.601,Z 440.782,A -85,B 0,C 180,E1 -23065.838,E2 -23065.838} C_VEL
LIN {X 0,Y 181.062,Z 442.899,A -85,B 0,C 180,E1 -23067.761,E2 -23067.761} C_VEL
LIN {X 0,Y 183.856,Z 447.609,A -85,B 0,C 180,E1 -23071.067,E2 -23071.067} C_VEL
LIN {X 0,Y 186.983,Z 453.038,A -85,B 0,C 180,E1 -23074.319,E2 -23074.319} C_VEL
LIN {X 0,Y 190.651,Z 459.892,A -85,B 0,C 180,E1 -23077.731,E2 -23077.731} C_VEL
LIN {X 0,Y 194.748,Z 468.172,A -85,B 0,C 180,E1 -23081.193,E2 -23081.193} C_VEL
LIN {X 0,Y 197.646,Z 474.379,A -85,B 0,C 180,E1 -23083.47,E2 -23083.47} C_VEL
LIN {X 0,Y 198.691,Z 480.749,A -85,B 0,C 180,E1 -23085.026,E2 -23085.026} C_VEL
LIN {X 0,Y 199.115,Z 485.494,A -85,B 0,C 180,E1 -23086.069,E2 -23086.069} C_VEL
LIN {X 0,Y 198.63,Z 488.882,A -85,B 0,C 180,E1 -23086.577,E2 -23086.577} C_VEL
LIN {X 0,Y 200.886,Z 518.18,A -85,B 0,C 180,E1 -23088.57,E2 -23088.57} C_VEL
LIN {X 0,Y 201.661,Z 531.29,A -85,B 0,C 180,E1 -23089.37,E2 -23089.37} C_VEL
LIN {X 0,Y 201.623,Z 535.162,A -85,B 0,C 180,E1 -23089.538,E2 -23089.538} C_VEL
LIN {X 0,Y 201.069,Z 539.05,A -85,B 0,C 180,E1 -23089.581,E2 -23089.581} C_VEL
LIN {X 0,Y 199.048,Z 546.724,A -85,B 0,C 180,E1 -23089.439,E2 -23089.439} C_VEL
LIN {X 0,Y 196.272,Z 556.382,A -85,B 0,C 180,E1 -23089.198,E2 -23089.198} C_VEL
LIN {X 0,Y 195.372,Z 562.311,A -85,B 0,C 180,E1 -23089.251,E2 -23089.251} C_VEL
LIN {X 0,Y 193.069,Z 602.841,A -85,B 0,C 180,E1 -23090.639,E2 -23090.639} C_VEL
LIN {X 0,Y 191.592,Z 615.725,A -85,B 0,C 180,E1 -23091.339,E2 -23091.339} C_VEL
LIN {X 0,Y 189.315,Z 628.286,A -85,B 0,C 180,E1 -23092.394,E2 -23092.394} C_VEL
LIN {X 0,Y 186.46,Z 640.839,A -85,B 0,C 180,E1 -23093.918,E2 -23093.918} C_VEL
LIN {X 0,Y 183.52,Z 651.304,A -85,B 0,C 180,E1 -23095.607,E2 -23095.607} C_VEL
LIN {X 0,Y 179.946,Z 661.999,A -85,B 0,C 180,E1 -23097.849,E2 -23097.849} C_VEL
LIN {X 0,Y 176.641,Z 670.726,A -85,B 0,C 180,E1 -23100.176,E2 -23100.176} C_VEL
LIN {X 0,Y 173.45,Z 678.736,A -85,B 0,C 180,E1 -23102.881,E2 -23102.881} C_VEL
LIN {X 0,Y 170.676,Z 685.371,A -85,B 0,C 180,E1 -23105.683,E2 -23105.683} C_VEL
LIN {X 0,Y 167.748,Z 691.891,A -85,B 0,C 180,E1 -23109.138,E2 -23109.138} C_VEL
LIN {X 0,Y 165.328,Z 697.067,A -85,B 0,C 180,E1 -23112.688,E2 -23112.688} C_VEL
LIN {X 0,Y 163.712,Z 701.065,A -85,B 0,C 180,E1 -23116.342,E2 -23116.342} C_VEL
LIN {X 0,Y 162.597,Z 704.009,A -85,B 0,C 180,E1 -23120.043,E2 -23120.043} C_VEL
LIN {X 0,Y 162.139,Z 705.419,A -85,B 0,C 180,E1 -23122.528,E2 -23122.528} C_VEL
LIN {X 0,Y 161.829,Z 706.975,A -85,B 0,C 180,E1 -23127.259,E2 -23127.259} C_VEL
LIN {X 0,Y 161.861,Z 707.237,A -85,B 0,C 180,E1 -23130,E2 -23130} C_VEL
LIN {X 0,Y 161.833,Z 706.956,A -85,B 0,C 180,E1 -23132.768,E2 -23132.768} C_VEL
LIN {X 0,Y 162.139,Z 705.387,A -85,B 0,C 180,E1 -23137.471,E2 -23137.471} C_VEL
LIN {X 0,Y 162.598,Z 703.958,A -85,B 0,C 180,E1 -23139.956,E2 -23139.956} C_VEL
LIN {X 0,Y 163.716,Z 700.995,A -85,B 0,C 180,E1 -23143.656,E2 -23143.656} C_VEL
LIN {X 0,Y 165.342,Z 696.972,A -85,B 0,C 180,E1 -23147.31,E2 -23147.31} C_VEL
LIN {X 0,Y 168.23,Z 690.773,A -85,B 0,C 180,E1 -23151.441,E2 -23151.441} C_VEL
LIN {X 0,Y 171.174,Z 684.156,A -85,B 0,C 180,E1 -23154.81,E2 -23154.81} C_VEL
LIN {X 0,Y 174.068,Z 677.088,A -85,B 0,C 180,E1 -23157.666,E2 -23157.666} C_VEL
LIN {X 0,Y 177.347,Z 668.728,A -85,B 0,C 180,E1 -23160.349,E2 -23160.349} C_VEL
LIN {X 0,Y 181.054,Z 658.389,A -85,B 0,C 180,E1 -23162.918,E2 -23162.918} C_VEL
LIN {X 0,Y 184.733,Z 646.752,A -85,B 0,C 180,E1 -23165.129,E2 -23165.129} C_VEL
LIN {X 0,Y 185.503,Z 644.58,A -85,B 0,C 180,E1 -23165.543,E2 -23165.543} C_VEL
LIN {X 0,Y 194.674,Z 639.43,A -85,B 0,C 180,E1 -23169.181,E2 -23169.181} C_VEL
LIN {X 0,Y 204.376,Z 633.306,A -85,B 0,C 180,E1 -23172.11,E2 -23172.11} C_VEL
LIN {X 0,Y 213.717,Z 626.708,A -85,B 0,C 180,E1 -23174.331,E2 -23174.331} C_VEL
LIN {X 0,Y 223.624,Z 618.799,A -85,B 0,C 180,E1 -23176.289,E2 -23176.289} C_VEL
LIN {X 0,Y 234.198,Z 609.251,A -85,B 0,C 180,E1 -23177.982,E2 -23177.982} C_VEL
LIN {X 0,Y 234.514,Z 608.72,A -85,B 0,C 180,E1 -23178.403,E2 -23178.403} C_VEL
LIN {X 0,Y 225.933,Z 614.728,A -85,B 0,C 180,E1 -23180.381,E2 -23180.381} C_VEL
LIN {X 0,Y 216.06,Z 620.303,A -85,B 0,C 180,E1 -23183.003,E2 -23183.003} C_VEL
LIN {X 0,Y 209.028,Z 623.383,A -85,B 0,C 180,E1 -23185.14,E2 -23185.14} C_VEL
LIN {X 0,Y 200.221,Z 626.138,A -85,B 0,C 180,E1 -23188.23,E2 -23188.23} C_VEL
LIN {X 0,Y 192.131,Z 627.397,A -85,B 0,C 180,E1 -23191.606,E2 -23191.606} C_VEL
LIN {X 0,Y 184.913,Z 627.218,A -85,B 0,C 180,E1 -23195.287,E2 -23195.287} C_VEL
LIN {X 0,Y 178.661,Z 625.515,A -85,B 0,C 180,E1 -23199.266,E2 -23199.266} C_VEL
LIN {X 0,Y 173.486,Z 622.341,A -85,B 0,C 180,E1 -23203.526,E2 -23203.526} C_VEL
LIN {X 0,Y 170.318,Z 618.948,A -85,B 0,C 180,E1 -23206.882,E2 -23206.882} C_VEL
LIN {X 0,Y 168.041,Z 614.629,A -85,B 0,C 180,E1 -23210.37,E2 -23210.37} C_VEL
LIN {X 0,Y 166.227,Z 609.338,A -85,B 0,C 180,E1 -23213.933,E2 -23213.933} C_VEL
LIN {X 0,Y 164.742,Z 601.742,A -85,B 0,C 180,E1 -23218.167,E2 -23218.167} C_VEL
LIN {X 0,Y 164.312,Z 593.796,A -85,B 0,C 180,E1 -23221.838,E2 -23221.838} C_VEL
LIN {X 0,Y 164.331,Z 584.272,A -85,B 0,C 180,E1 -23225.522,E2 -23225.522} C_VEL
LIN {X 0,Y 164.777,Z 574.805,A -85,B 0,C 180,E1 -23228.585,E2 -23228.585} C_VEL
LIN {X 0,Y 165.362,Z 564.769,A -85,B 0,C 180,E1 -23231.296,E2 -23231.296} C_VEL
LIN {X 0,Y 166.108,Z 552.531,A -85,B 0,C 180,E1 -23234.018,E2 -23234.018} C_VEL
LIN {X 0,Y 166.823,Z 540.469,A -85,B 0,C 180,E1 -23236.207,E2 -23236.207} C_VEL
LIN {X 0,Y 167.675,Z 526.776,A -85,B 0,C 180,E1 -23238.164,E2 -23238.164} C_VEL
LIN {X 0,Y 168.273,Z 514.439,A -85,B 0,C 180,E1 -23239.519,E2 -23239.519} C_VEL
LIN {X 0,Y 169.852,Z 462.606,A -85,B 0,C 180,E1 -23243.631,E2 -23243.631} C_VEL
LIN {X 0,Y 170.047,Z 460.541,A -85,B 0,C 180,E1 -23244.088,E2 -23244.088} C_VEL
LIN {X 0,Y 170.234,Z 460.135,A -85,B 0,C 180,E1 -23244.384,E2 -23244.384} C_VEL
LIN {X 0,Y 171.631,Z 459.647,A -85,B 0,C 180,E1 -23245.253,E2 -23245.253} C_VEL
LIN {X 0,Y 173.145,Z 458.622,A -85,B 0,C 180,E1 -23245.765,E2 -23245.765} C_VEL
LIN {X 0,Y 175.191,Z 456.793,A -85,B 0,C 180,E1 -23246.186,E2 -23246.186} C_VEL
LIN {X 0,Y 178.922,Z 456.198,A -85,B 0,C 180,E1 -23248.123,E2 -23248.123} C_VEL
LIN {X 0,Y 181.872,Z 463.793,A -85,B 0,C 180,E1 -23252.752,E2 -23252.752} C_VEL
LIN {X 0,Y 184.126,Z 470.634,A -85,B 0,C 180,E1 -23256.274,E2 -23256.274} C_VEL
LIN {X 0,Y 186.995,Z 480.399,A -85,B 0,C 180,E1 -23260.5,E2 -23260.5} C_VEL
LIN {X 0,Y 188.766,Z 488.384,A -85,B 0,C 180,E1 -23263.64,E2 -23263.64} C_VEL
LIN {X 0,Y 193.647,Z 499.28,A -85,B 0,C 180,E1 -23265.701,E2 -23265.701} C_VEL
LIN {X 0,Y 196.061,Z 523.574,A -85,B 0,C 180,E1 -23267.579,E2 -23267.579} C_VEL
LIN {X 0,Y 197.074,Z 537.088,A -85,B 0,C 180,E1 -23268.495,E2 -23268.495} C_VEL
LIN {X 0,Y 193.261,Z 602.594,A -85,B 0,C 180,E1 -23270.738,E2 -23270.738} C_VEL
LIN {X 0,Y 191.534,Z 615.397,A -85,B 0,C 180,E1 -23271.491,E2 -23271.491} C_VEL
LIN {X 0,Y 189.197,Z 628.388,A -85,B 0,C 180,E1 -23272.703,E2 -23272.703} C_VEL
LIN {X 0,Y 186.381,Z 640.26,A -85,B 0,C 180,E1 -23274.235,E2 -23274.235} C_VEL
LIN {X 0,Y 183.055,Z 651.53,A -85,B 0,C 180,E1 -23276.173,E2 -23276.173} C_VEL
LIN {X 0,Y 179.572,Z 661.706,A -85,B 0,C 180,E1 -23278.435,E2 -23278.435} C_VEL
LIN {X 0,Y 176.477,Z 670.047,A -85,B 0,C 180,E1 -23280.801,E2 -23280.801} C_VEL
LIN {X 0,Y 173.397,Z 677.74,A -85,B 0,C 180,E1 -23283.523,E2 -23283.523} C_VEL
LIN {X 0,Y 170.086,Z 685.233,A -85,B 0,C 180,E1 -23286.887,E2 -23286.887} C_VEL
LIN {X 0,Y 167.222,Z 691.244,A -85,B 0,C 180,E1 -23290.353,E2 -23290.353} C_VEL
LIN {X 0,Y 165.113,Z 695.996,A -85,B 0,C 180,E1 -23293.939,E2 -23293.939} C_VEL
LIN {X 0,Y 163.545,Z 699.63,A -85,B 0,C 180,E1 -23297.593,E2 -23297.593} C_VEL
LIN {X 0,Y 162.781,Z 701.501,A -85,B 0,C 180,E1 -23300.056,E2 -23300.056} C_VEL
LIN {X 0,Y 162.254,Z 702.925,A -85,B 0,C 180,E1 -23302.534,E2 -23302.534} C_VEL
LIN {X 0,Y 161.936,Z 703.924,A -85,B 0,C 180,E1 -23305.021,E2 -23305.021} C_VEL
LIN {X 0,Y 161.798,Z 704.539,A -85,B 0,C 180,E1 -23307.511,E2 -23307.511} C_VEL
LIN {X 0,Y 161.782,Z 704.77,A -85,B 0,C 180,E1 -23310,E2 -23310} C_VEL
LIN {X 0,Y 161.798,Z 704.57,A -85,B 0,C 180,E1 -23312.49,E2 -23312.49} C_VEL
LIN {X 0,Y 161.935,Z 703.975,A -85,B 0,C 180,E1 -23314.98,E2 -23314.98} C_VEL
LIN {X 0,Y 162.208,Z 702.997,A -85,B 0,C 180,E1 -23317.469,E2 -23317.469} C_VEL
LIN {X 0,Y 162.716,Z 701.614,A -85,B 0,C 180,E1 -23319.949,E2 -23319.949} C_VEL
LIN {X 0,Y 163.926,Z 698.711,A -85,B 0,C 180,E1 -23323.639,E2 -23323.639} C_VEL
LIN {X 0,Y 165.657,Z 694.767,A -85,B 0,C 180,E1 -23327.276,E2 -23327.276} C_VEL
LIN {X 0,Y 168.076,Z 689.655,A -85,B 0,C 180,E1 -23330.82,E2 -23330.82} C_VEL
LIN {X 0,Y 171.045,Z 683.212,A -85,B 0,C 180,E1 -23334.261,E2 -23334.261} C_VEL
LIN {X 0,Y 174.466,Z 675.21,A -85,B 0,C 180,E1 -23337.597,E2 -23337.597} C_VEL
LIN {X 0,Y 177.662,Z 667.017,A -85,B 0,C 180,E1 -23340.29,E2 -23340.29} C_VEL
LIN {X 0,Y 180.987,Z 658.057,A -85,B 0,C 180,E1 -23342.602,E2 -23342.602} C_VEL
LIN {X 0,Y 184.589,Z 646.939,A -85,B 0,C 180,E1 -23344.828,E2 -23344.828} C_VEL
LIN {X 0,Y 187.547,Z 636.081,A -85,B 0,C 180,E1 -23346.505,E2 -23346.505} C_VEL
LIN {X 0,Y 190.178,Z 624.033,A -85,B 0,C 180,E1 -23347.907,E2 -23347.907} C_VEL
LIN {X 0,Y 192.331,Z 611.454,A -85,B 0,C 180,E1 -23348.907,E2 -23348.907} C_VEL
LIN {X 0,Y 193.688,Z 598.53,A -85,B 0,C 180,E1 -23349.588,E2 -23349.588} C_VEL
LIN {X 0,Y 197.21,Z 535.592,A -85,B 0,C 180,E1 -23351.717,E2 -23351.717} C_VEL
LIN {X 0,Y 194.84,Z 509.243,A -85,B 0,C 180,E1 -23353.642,E2 -23353.642} C_VEL
LIN {X 0,Y 193.669,Z 499.079,A -85,B 0,C 180,E1 -23354.488,E2 -23354.488} C_VEL
LIN {X 0,Y 188.65,Z 487.986,A -85,B 0,C 180,E1 -23356.645,E2 -23356.645} C_VEL
LIN {X 0,Y 186.54,Z 479.027,A -85,B 0,C 180,E1 -23360.172,E2 -23360.172} C_VEL
LIN {X 0,Y 184.27,Z 471.068,A -85,B 0,C 180,E1 -23363.759,E2 -23363.759} C_VEL
LIN {X 0,Y 182.054,Z 464.234,A -85,B 0,C 180,E1 -23367.285,E2 -23367.285} C_VEL
LIN {X 0,Y 179.818,Z 458.215,A -85,B 0,C 180,E1 -23370.84,E2 -23370.84} C_VEL
LIN {X 0,Y 177.801,Z 453.215,A -85,B 0,C 180,E1 -23374.227,E2 -23374.227} C_VEL
LIN {X 0,Y 175.112,Z 447.564,A -85,B 0,C 180,E1 -23378.825,E2 -23378.825} C_VEL
LIN {X 0,Y 172.905,Z 442.789,A -85,B 0,C 180,E1 -23383.469,E2 -23383.469} C_VEL
LIN {X 0,Y 170.42,Z 437.726,A -85,B 0,C 180,E1 -23390.505,E2 -23390.505} C_VEL
LIN {X 0,Y 168.881,Z 434.212,A -85,B 0,C 180,E1 -23400,E2 -23400} C_VEL
LIN {X 0,Y 168.656,Z 434.161,A -85,B 0,C 180,E1 -23402.388,E2 -23402.388} C_VEL
LIN {X 0,Y 168.746,Z 434.946,A -85,B 0,C 180,E1 -23407.177,E2 -23407.177} C_VEL
LIN {X 0,Y 170.323,Z 437.621,A -85,B 0,C 180,E1 -23414.334,E2 -23414.334} C_VEL
LIN {X 0,Y 171.249,Z 438.718,A -85,B 0,C 180,E1 -23416.695,E2 -23416.695} C_VEL
LIN {X 0,Y 174.046,Z 443.358,A -85,B 0,C 180,E1 -23422.558,E2 -23422.558} C_VEL
LIN {X 0,Y 177.021,Z 448.451,A -85,B 0,C 180,E1 -23427.166,E2 -23427.166} C_VEL
LIN {X 0,Y 180.056,Z 453.645,A -85,B 0,C 180,E1 -23430.827,E2 -23430.827} C_VEL
LIN {X 0,Y 183.117,Z 459.114,A -85,B 0,C 180,E1 -23434.136,E2 -23434.136} C_VEL
LIN {X 0,Y 187.341,Z 467.401,A -85,B 0,C 180,E1 -23438.241,E2 -23438.241} C_VEL
LIN {X 0,Y 191.658,Z 476.727,A -85,B 0,C 180,E1 -23442.008,E2 -23442.008} C_VEL
LIN {X 0,Y 192.705,Z 479.128,A -85,B 0,C 180,E1 -23442.867,E2 -23442.867} C_VEL
LIN {X 0,Y 193.567,Z 487.247,A -85,B 0,C 180,E1 -23444.849,E2 -23444.849} C_VEL
LIN {X 0,Y 193.477,Z 489.34,A -85,B 0,C 180,E1 -23445.136,E2 -23445.136} C_VEL
LIN {X 0,Y 195.667,Z 520.458,A -85,B 0,C 180,E1 -23447.314,E2 -23447.314} C_VEL
LIN {X 0,Y 196.646,Z 540.478,A -85,B 0,C 180,E1 -23448.539,E2 -23448.539} C_VEL
LIN {X 0,Y 195.372,Z 562.311,A -85,B 0,C 180,E1 -23449.251,E2 -23449.251} C_VEL
LIN {X 0,Y 194.516,Z 568.158,A -85,B 0,C 180,E1 -23449.312,E2 -23449.312} C_VEL
LIN {X 0,Y 189.153,Z 587.184,A -85,B 0,C 180,E1 -23448.841,E2 -23448.841} C_VEL
LIN {X 0,Y 188.357,Z 593.027,A -85,B 0,C 180,E1 -23448.918,E2 -23448.918} C_VEL
LIN {X 0,Y 187.053,Z 608.755,A -85,B 0,C 180,E1 -23449.551,E2 -23449.551} C_VEL
LIN {X 0,Y 185.183,Z 620.887,A -85,B 0,C 180,E1 -23450.352,E2 -23450.352} C_VEL
LIN {X 0,Y 182.598,Z 633.527,A -85,B 0,C 180,E1 -23451.637,E2 -23451.637} C_VEL
LIN {X 0,Y 179.446,Z 645.565,A -85,B 0,C 180,E1 -23453.325,E2 -23453.325} C_VEL
LIN {X 0,Y 176.008,Z 656.326,A -85,B 0,C 180,E1 -23455.319,E2 -23455.319} C_VEL
LIN {X 0,Y 171.996,Z 667.008,A -85,B 0,C 180,E1 -23457.913,E2 -23457.913} C_VEL
LIN {X 0,Y 168.434,Z 675.682,A -85,B 0,C 180,E1 -23460.641,E2 -23460.641} C_VEL
LIN {X 0,Y 165.007,Z 683.738,A -85,B 0,C 180,E1 -23463.912,E2 -23463.912} C_VEL
LIN {X 0,Y 161.625,Z 690.84,A -85,B 0,C 180,E1 -23467.636,E2 -23467.636} C_VEL
LIN {X 0,Y 158.534,Z 697.015,A -85,B 0,C 180,E1 -23471.921,E2 -23471.921} C_VEL
LIN {X 0,Y 156.796,Z 701.012,A -85,B 0,C 180,E1 -23475.728,E2 -23475.728} C_VEL
LIN {X 0,Y 155.576,Z 703.956,A -85,B 0,C 180,E1 -23479.589,E2 -23479.589} C_VEL
LIN {X 0,Y 155.077,Z 705.365,A -85,B 0,C 180,E1 -23482.186,E2 -23482.186} C_VEL
LIN {X 0,Y 154.851,Z 706.362,A -85,B 0,C 180,E1 -23484.792,E2 -23484.792} C_VEL
LIN {X 0,Y 154.742,Z 707.024,A -85,B 0,C 180,E1 -23487.69,E2 -23487.69} C_VEL
LIN {X 0,Y 154.774,Z 707.183,A -85,B 0,C 180,E1 -23490,E2 -23490} C_VEL
LIN {X 0,Y 154.739,Z 706.955,A -85,B 0,C 180,E1 -23492.603,E2 -23492.603} C_VEL
LIN {X 0,Y 154.851,Z 706.338,A -85,B 0,C 180,E1 -23495.208,E2 -23495.208} C_VEL
LIN {X 0,Y 155.077,Z 705.333,A -85,B 0,C 180,E1 -23497.814,E2 -23497.814} C_VEL
LIN {X 0,Y 155.578,Z 703.904,A -85,B 0,C 180,E1 -23500.41,E2 -23500.41} C_VEL
LIN {X 0,Y 156.8,Z 700.94,A -85,B 0,C 180,E1 -23504.271,E2 -23504.271} C_VEL
LIN {X 0,Y 158.549,Z 696.917,A -85,B 0,C 180,E1 -23508.076,E2 -23508.076} C_VEL
LIN {X 0,Y 161.627,Z 690.719,A -85,B 0,C 180,E1 -23512.363,E2 -23512.363} C_VEL
LIN {X 0,Y 165,Z 683.595,A -85,B 0,C 180,E1 -23516.087,E2 -23516.087} C_VEL
LIN {X 0,Y 168.431,Z 675.479,A -85,B 0,C 180,E1 -23519.359,E2 -23519.359} C_VEL
LIN {X 0,Y 172.011,Z 666.756,A -85,B 0,C 180,E1 -23522.083,E2 -23522.083} C_VEL
LIN {X 0,Y 175.982,Z 656.024,A -85,B 0,C 180,E1 -23524.686,E2 -23524.686} C_VEL
LIN {X 0,Y 179.918,Z 644.213,A -85,B 0,C 180,E1 -23526.911,E2 -23526.911} C_VEL
LIN {X 0,Y 189.239,Z 639.706,A -85,B 0,C 180,E1 -23530.535,E2 -23530.535} C_VEL
LIN {X 0,Y 199.191,Z 634.22,A -85,B 0,C 180,E1 -23533.473,E2 -23533.473} C_VEL
LIN {X 0,Y 210.121,Z 627.318,A -85,B 0,C 180,E1 -23535.982,E2 -23535.982} C_VEL
LIN {X 0,Y 219.365,Z 620.672,A -85,B 0,C 180,E1 -23537.717,E2 -23537.717} C_VEL
LIN {X 0,Y 223.449,Z 617.483,A -85,B 0,C 180,E1 -23538.383,E2 -23538.383} C_VEL
LIN {X 0,Y 223.719,Z 617.094,A -85,B 0,C 180,E1 -23538.723,E2 -23538.723} C_VEL
LIN {X 0,Y 213.406,Z 622.431,A -85,B 0,C 180,E1 -23541.265,E2 -23541.265} C_VEL
LIN {X 0,Y 203.617,Z 626.133,A -85,B 0,C 180,E1 -23544.072,E2 -23544.072} C_VEL
LIN {X 0,Y 194.479,Z 628.36,A -85,B 0,C 180,E1 -23547.176,E2 -23547.176} C_VEL
LIN {X 0,Y 186.076,Z 629.093,A -85,B 0,C 180,E1 -23550.593,E2 -23550.593} C_VEL
LIN {X 0,Y 178.585,Z 628.397,A -85,B 0,C 180,E1 -23554.349,E2 -23554.349} C_VEL
LIN {X 0,Y 172.088,Z 626.247,A -85,B 0,C 180,E1 -23558.435,E2 -23558.435} C_VEL
LIN {X 0,Y 166.708,Z 622.58,A -85,B 0,C 180,E1 -23562.836,E2 -23562.836} C_VEL
LIN {X 0,Y 162.508,Z 617.413,A -85,B 0,C 180,E1 -23567.512,E2 -23567.512} C_VEL
LIN {X 0,Y 160.431,Z 612.436,A -85,B 0,C 180,E1 -23571.18,E2 -23571.18} C_VEL
LIN {X 0,Y 158.442,Z 605.241,A -85,B 0,C 180,E1 -23575.548,E2 -23575.548} C_VEL
LIN {X 0,Y 157.435,Z 596.459,A -85,B 0,C 180,E1 -23580,E2 -23580} C_VEL
LIN {X 0,Y 157.266,Z 587.223,A -85,B 0,C 180,E1 -23583.844,E2 -23583.844} C_VEL
LIN {X 0,Y 157.66,Z 576.105,A -85,B 0,C 180,E1 -23587.685,E2 -23587.685} C_VEL
LIN {X 0,Y 158.331,Z 564.376,A -85,B 0,C 180,E1 -23591.007,E2 -23591.007} C_VEL
LIN {X 0,Y 159.076,Z 551.508,A -85,B 0,C 180,E1 -23593.933,E2 -23593.933} C_VEL
LIN {X 0,Y 159.878,Z 538.521,A -85,B 0,C 180,E1 -23596.274,E2 -23596.274} C_VEL
LIN {X 0,Y 160.758,Z 523.999,A -85,B 0,C 180,E1 -23598.314,E2 -23598.314} C_VEL
LIN {X 0,Y 161.342,Z 510.286,A -85,B 0,C 180,E1 -23599.73,E2 -23599.73} C_VEL
LIN {X 0,Y 162.394,Z 471.483,A -85,B 0,C 180,E1 -23603.008,E2 -23603.008} C_VEL
LIN {X 0,Y 162.56,Z 469.661,A -85,B 0,C 180,E1 -23603.488,E2 -23603.488} C_VEL
LIN {X 0,Y 163.16,Z 469.199,A -85,B 0,C 180,E1 -23604.155,E2 -23604.155} C_VEL
LIN {X 0,Y 165.362,Z 467.982,A -85,B 0,C 180,E1 -23605.151,E2 -23605.151} C_VEL
LIN {X 0,Y 168.301,Z 465.662,A -85,B 0,C 180,E1 -23606.006,E2 -23606.006} C_VEL
LIN {X 0,Y 170.578,Z 464.526,A -85,B 0,C 180,E1 -23606.95,E2 -23606.95} C_VEL
LIN {X 0,Y 173.48,Z 462.407,A -85,B 0,C 180,E1 -23607.768,E2 -23607.768} C_VEL
LIN {X 0,Y 174.87,Z 463.009,A -85,B 0,C 180,E1 -23608.835,E2 -23608.835} C_VEL
LIN {X 0,Y 177.279,Z 469.728,A -85,B 0,C 180,E1 -23612.86,E2 -23612.86} C_VEL
LIN {X 0,Y 179.541,Z 477.016,A -85,B 0,C 180,E1 -23616.555,E2 -23616.555} C_VEL
LIN {X 0,Y 181.436,Z 484.07,A -85,B 0,C 180,E1 -23619.726,E2 -23619.726} C_VEL
LIN {X 0,Y 182.48,Z 488.591,A -85,B 0,C 180,E1 -23621.549,E2 -23621.549} C_VEL
LIN {X 0,Y 187.079,Z 498.418,A -85,B 0,C 180,E1 -23623.66,E2 -23623.66} C_VEL
LIN {X 0,Y 188.77,Z 502.385,A -85,B 0,C 180,E1 -23624.407,E2 -23624.407} C_VEL
LIN {X 0,Y 190.88,Z 525.146,A -85,B 0,C 180,E1 -23626.224,E2 -23626.224} C_VEL
LIN {X 0,Y 191.777,Z 537.447,A -85,B 0,C 180,E1 -23627.099,E2 -23627.099} C_VEL
LIN {X 0,Y 187.914,Z 601.62,A -85,B 0,C 180,E1 -23629.328,E2 -23629.328} C_VEL
LIN {X 0,Y 186.193,Z 614.705,A -85,B 0,C 180,E1 -23630.083,E2 -23630.083} C_VEL
LIN {X 0,Y 184.074,Z 626.259,A -85,B 0,C 180,E1 -23631.128,E2 -23631.128} C_VEL
LIN {X 0,Y 181.125,Z 638.653,A -85,B 0,C 180,E1 -23632.679,E2 -23632.679} C_VEL
LIN {X 0,Y 178.064,Z 649.035,A -85,B 0,C 180,E1 -23634.397,E2 -23634.397} C_VEL
LIN {X 0,Y 174.344,Z 659.666,A -85,B 0,C 180,E1 -23636.685,E2 -23636.685} C_VEL
LIN {X 0,Y 170.955,Z 668.351,A -85,B 0,C 180,E1 -23639.078,E2 -23639.078} C_VEL
LIN {X 0,Y 167.713,Z 676.286,A -85,B 0,C 180,E1 -23641.849,E2 -23641.849} C_VEL
LIN {X 0,Y 164.114,Z 684.166,A -85,B 0,C 180,E1 -23645.321,E2 -23645.321} C_VEL
LIN {X 0,Y 161.515,Z 689.452,A -85,B 0,C 180,E1 -23648.293,E2 -23648.293} C_VEL
LIN {X 0,Y 158.951,Z 694.616,A -85,B 0,C 180,E1 -23651.971,E2 -23651.971} C_VEL
LIN {X 0,Y 157.073,Z 698.611,A -85,B 0,C 180,E1 -23655.754,E2 -23655.754} C_VEL
LIN {X 0,Y 155.79,Z 701.555,A -85,B 0,C 180,E1 -23659.604,E2 -23659.604} C_VEL
LIN {X 0,Y 155.211,Z 702.979,A -85,B 0,C 180,E1 -23662.193,E2 -23662.193} C_VEL
LIN {X 0,Y 154.861,Z 703.978,A -85,B 0,C 180,E1 -23664.793,E2 -23664.793} C_VEL
LIN {X 0,Y 154.653,Z 704.751,A -85,B 0,C 180,E1 -23668.764,E2 -23668.764} C_VEL
LIN {X 0,Y 154.701,Z 704.623,A -85,B 0,C 180,E1 -23672.604,E2 -23672.604} C_VEL
LIN {X 0,Y 154.859,Z 704.029,A -85,B 0,C 180,E1 -23675.208,E2 -23675.208} C_VEL
LIN {X 0,Y 155.174,Z 703.051,A -85,B 0,C 180,E1 -23677.81,E2 -23677.81} C_VEL
LIN {X 0,Y 155.709,Z 701.667,A -85,B 0,C 180,E1 -23680.402,E2 -23680.402} C_VEL
LIN {X 0,Y 157.015,Z 698.764,A -85,B 0,C 180,E1 -23684.252,E2 -23684.252} C_VEL
LIN {X 0,Y 158.862,Z 694.819,A -85,B 0,C 180,E1 -23688.04,E2 -23688.04} C_VEL
LIN {X 0,Y 161.46,Z 689.706,A -85,B 0,C 180,E1 -23691.715,E2 -23691.715} C_VEL
LIN {X 0,Y 164.57,Z 683.262,A -85,B 0,C 180,E1 -23695.281,E2 -23695.281} C_VEL
LIN {X 0,Y 167.976,Z 675.763,A -85,B 0,C 180,E1 -23698.523,E2 -23698.523} C_VEL
LIN {X 0,Y 171.566,Z 667.062,A -85,B 0,C 180,E1 -23701.487,E2 -23701.487} C_VEL
LIN {X 0,Y 175.065,Z 658.098,A -85,B 0,C 180,E1 -23703.85,E2 -23703.85} C_VEL
LIN {X 0,Y 178.814,Z 646.975,A -85,B 0,C 180,E1 -23706.126,E2 -23706.126} C_VEL
LIN {X 0,Y 181.897,Z 636.111,A -85,B 0,C 180,E1 -23707.834,E2 -23707.834} C_VEL
LIN {X 0,Y 184.642,Z 624.05,A -85,B 0,C 180,E1 -23709.257,E2 -23709.257} C_VEL
LIN {X 0,Y 186.874,Z 611.45,A -85,B 0,C 180,E1 -23710.271,E2 -23710.271} C_VEL
LIN {X 0,Y 188.28,Z 598.485,A -85,B 0,C 180,E1 -23710.963,E2 -23710.963} C_VEL
LIN {X 0,Y 191.926,Z 536.682,A -85,B 0,C 180,E1 -23713.08,E2 -23713.08} C_VEL
LIN {X 0,Y 189.782,Z 511.209,A -85,B 0,C 180,E1 -23715.008,E2 -23715.008} C_VEL
LIN {X 0,Y 188.74,Z 501.967,A -85,B 0,C 180,E1 -23715.817,E2 -23715.817} C_VEL
LIN {X 0,Y 183.771,Z 491.22,A -85,B 0,C 180,E1 -23718.042,E2 -23718.042} C_VEL
LIN {X 0,Y 182.3,Z 487.901,A -85,B 0,C 180,E1 -23718.824,E2 -23718.824} C_VEL
LIN {X 0,Y 180.021,Z 478.749,A -85,B 0,C 180,E1 -23722.777,E2 -23722.777} C_VEL
LIN {X 0,Y 177.54,Z 470.305,A -85,B 0,C 180,E1 -23727.042,E2 -23727.042} C_VEL
LIN {X 0,Y 175.838,Z 465.204,A -85,B 0,C 180,E1 -23730.026,E2 -23730.026} C_VEL
LIN {X 0,Y 173.149,Z 458.297,A -85,B 0,C 180,E1 -23734.774,E2 -23734.774} C_VEL
LIN {X 0,Y 170.626,Z 452.721,A -85,B 0,C 180,E1 -23739.506,E2 -23739.506} C_VEL
LIN {X 0,Y 169.095,Z 449.262,A -85,B 0,C 180,E1 -23743.086,E2 -23743.086} C_VEL
LIN {X 0,Y 167.242,Z 445.533,A -85,B 0,C 180,E1 -23747.871,E2 -23747.871} C_VEL
LIN {X 0,Y 166.629,Z 443.928,A -85,B 0,C 180,E1 -23750.287,E2 -23750.287} C_VEL
LIN {X 0,Y 165.288,Z 441.207,A -85,B 0,C 180,E1 -23757.563,E2 -23757.563} C_VEL
LIN {X 0,Y 165.251,Z 440.334,A -85,B 0,C 180,E1 -23760,E2 -23760} C_VEL
LIN {X 0,Y 165.036,Z 440.282,A -85,B 0,C 180,E1 -23762.441,E2 -23762.441} C_VEL
LIN {X 0,Y 165.208,Z 441.154,A -85,B 0,C 180,E1 -23767.332,E2 -23767.332} C_VEL
LIN {X 0,Y 166.893,Z 443.915,A -85,B 0,C 180,E1 -23774.635,E2 -23774.635} C_VEL
LIN {X 0,Y 167.807,Z 445.273,A -85,B 0,C 180,E1 -23777.048,E2 -23777.048} C_VEL
LIN {X 0,Y 170.039,Z 449.018,A -85,B 0,C 180,E1 -23781.838,E2 -23781.838} C_VEL
LIN {X 0,Y 173.051,Z 454.156,A -85,B 0,C 180,E1 -23786.686,E2 -23786.686} C_VEL
LIN {X 0,Y 175.66,Z 458.671,A -85,B 0,C 180,E1 -23790.008,E2 -23790.008} C_VEL
LIN {X 0,Y 178.635,Z 464.176,A -85,B 0,C 180,E1 -23793.422,E2 -23793.422} C_VEL
LIN {X 0,Y 183.025,Z 473.008,A -85,B 0,C 180,E1 -23797.907,E2 -23797.907} C_VEL
LIN {X 0,Y 187.264,Z 482.392,A -85,B 0,C 180,E1 -23801.708,E2 -23801.708} C_VEL
LIN {X 0,Y 187.717,Z 484.509,A -85,B 0,C 180,E1 -23802.37,E2 -23802.37} C_VEL
LIN {X 0,Y 188.153,Z 488.944,A -85,B 0,C 180,E1 -23803.471,E2 -23803.471} C_VEL
LIN {X 0,Y 188.524,Z 491.678,A -85,B 0,C 180,E1 -23803.739,E2 -23803.739} C_VEL
LIN {X 0,Y 190.268,Z 517.416,A -85,B 0,C 180,E1 -23805.633,E2 -23805.633} C_VEL
LIN {X 0,Y 191.337,Z 541.52,A -85,B 0,C 180,E1 -23807.167,E2 -23807.167} C_VEL
LIN {X 0,Y 188.357,Z 593.027,A -85,B 0,C 180,E1 -23808.918,E2 -23808.918} C_VEL
LIN {X 0,Y 187.493,Z 598.87,A -85,B 0,C 180,E1 -23808.982,E2 -23808.982} C_VEL
LIN {X 0,Y 184.412,Z 608.299,A -85,B 0,C 180,E1 -23808.809,E2 -23808.809} C_VEL
LIN {X 0,Y 180.896,Z 617.582,A -85,B 0,C 180,E1 -23808.795,E2 -23808.795} C_VEL
LIN {X 0,Y 179.337,Z 623.194,A -85,B 0,C 180,E1 -23809.12,E2 -23809.12} C_VEL
LIN {X 0,Y 176.588,Z 635.442,A -85,B 0,C 180,E1 -23810.447,E2 -23810.447} C_VEL
LIN {X 0,Y 173.337,Z 647.033,A -85,B 0,C 180,E1 -23812.175,E2 -23812.175} C_VEL
LIN {X 0,Y 169.327,Z 658.598,A -85,B 0,C 180,E1 -23814.473,E2 -23814.473} C_VEL
LIN {X 0,Y 165.241,Z 668.871,A -85,B 0,C 180,E1 -23817.16,E2 -23817.16} C_VEL
LIN {X 0,Y 161.566,Z 677.171,A -85,B 0,C 180,E1 -23819.983,E2 -23819.983} C_VEL
LIN {X 0,Y 157.846,Z 685.272,A -85,B 0,C 180,E1 -23823.56,E2 -23823.56} C_VEL
LIN {X 0,Y 154.551,Z 691.789,A -85,B 0,C 180,E1 -23827.261,E2 -23827.261} C_VEL
LIN {X 0,Y 151.779,Z 696.963,A -85,B 0,C 180,E1 -23831.087,E2 -23831.087} C_VEL
LIN {X 0,Y 149.906,Z 700.959,A -85,B 0,C 180,E1 -23835.057,E2 -23835.057} C_VEL
LIN {X 0,Y 148.58,Z 703.902,A -85,B 0,C 180,E1 -23839.093,E2 -23839.093} C_VEL
LIN {X 0,Y 148.028,Z 705.312,A -85,B 0,C 180,E1 -23841.811,E2 -23841.811} C_VEL
LIN {X 0,Y 147.759,Z 706.308,A -85,B 0,C 180,E1 -23844.541,E2 -23844.541} C_VEL
LIN {X 0,Y 147.63,Z 707.057,A -85,B 0,C 180,E1 -23848.637,E2 -23848.637} C_VEL
LIN {X 0,Y 147.646,Z 706.901,A -85,B 0,C 180,E1 -23852.728,E2 -23852.728} C_VEL
LIN {X 0,Y 147.759,Z 706.284,A -85,B 0,C 180,E1 -23855.458,E2 -23855.458} C_VEL
LIN {X 0,Y 148.029,Z 705.278,A -85,B 0,C 180,E1 -23858.188,E2 -23858.188} C_VEL
LIN {X 0,Y 148.581,Z 703.849,A -85,B 0,C 180,E1 -23860.906,E2 -23860.906} C_VEL
LIN {X 0,Y 149.91,Z 700.886,A -85,B 0,C 180,E1 -23864.942,E2 -23864.942} C_VEL
LIN {X 0,Y 151.794,Z 696.863,A -85,B 0,C 180,E1 -23868.911,E2 -23868.911} C_VEL
LIN {X 0,Y 155.067,Z 690.666,A -85,B 0,C 180,E1 -23873.364,E2 -23873.364} C_VEL
LIN {X 0,Y 158.501,Z 683.81,A -85,B 0,C 180,E1 -23877.087,E2 -23877.087} C_VEL
LIN {X 0,Y 161.564,Z 676.984,A -85,B 0,C 180,E1 -23880.016,E2 -23880.016} C_VEL
LIN {X 0,Y 165.226,Z 668.627,A -85,B 0,C 180,E1 -23882.842,E2 -23882.842} C_VEL
LIN {X 0,Y 169.31,Z 658.294,A -85,B 0,C 180,E1 -23885.53,E2 -23885.53} C_VEL
LIN {X 0,Y 173.301,Z 646.662,A -85,B 0,C 180,E1 -23887.834,E2 -23887.834} C_VEL
LIN {X 0,Y 174.444,Z 643.729,A -85,B 0,C 180,E1 -23888.366,E2 -23888.366} C_VEL
LIN {X 0,Y 183.918,Z 639.795,A -85,B 0,C 180,E1 -23891.969,E2 -23891.969} C_VEL
LIN {X 0,Y 194.11,Z 634.926,A -85,B 0,C 180,E1 -23894.912,E2 -23894.912} C_VEL
LIN {X 0,Y 205.262,Z 628.717,A -85,B 0,C 180,E1 -23897.404,E2 -23897.404} C_VEL
LIN {X 0,Y 212.382,Z 624.273,A -85,B 0,C 180,E1 -23898.724,E2 -23898.724} C_VEL
LIN {X 0,Y 211.767,Z 624.282,A -85,B 0,C 180,E1 -23899.292,E2 -23899.292} C_VEL
LIN {X 0,Y 203.214,Z 627.377,A -85,B 0,C 180,E1 -23901.5,E2 -23901.5} C_VEL
LIN {X 0,Y 193.437,Z 629.743,A -85,B 0,C 180,E1 -23904.457,E2 -23904.457} C_VEL
LIN {X 0,Y 184.321,Z 630.708,A -85,B 0,C 180,E1 -23907.737,E2 -23907.737} C_VEL
LIN {X 0,Y 176.075,Z 630.198,A -85,B 0,C 180,E1 -23911.381,E2 -23911.381} C_VEL
LIN {X 0,Y 168.759,Z 628.283,A -85,B 0,C 180,E1 -23915.389,E2 -23915.389} C_VEL
LIN {X 0,Y 162.574,Z 624.925,A -85,B 0,C 180,E1 -23919.767,E2 -23919.767} C_VEL
LIN {X 0,Y 157.594,Z 620.015,A -85,B 0,C 180,E1 -23924.48,E2 -23924.48} C_VEL
LIN {X 0,Y 154.833,Z 615.3,A -85,B 0,C 180,E1 -23928.214,E2 -23928.214} C_VEL
LIN {X 0,Y 152.465,Z 608.581,A -85,B 0,C 180,E1 -23932.718,E2 -23932.718} C_VEL
LIN {X 0,Y 150.833,Z 600.205,A -85,B 0,C 180,E1 -23937.329,E2 -23937.329} C_VEL
LIN {X 0,Y 150.332,Z 591.593,A -85,B 0,C 180,E1 -23941.34,E2 -23941.34} C_VEL
LIN {X 0,Y 150.4,Z 581.266,A -85,B 0,C 180,E1 -23945.363,E2 -23945.363} C_VEL
LIN {X 0,Y 150.893,Z 570.854,A -85,B 0,C 180,E1 -23948.707,E2 -23948.707} C_VEL
LIN {X 0,Y 151.558,Z 559.283,A -85,B 0,C 180,E1 -23951.787,E2 -23951.787} C_VEL
LIN {X 0,Y 152.264,Z 547.709,A -85,B 0,C 180,E1 -23954.33,E2 -23954.33} C_VEL
LIN {X 0,Y 153.106,Z 533.228,A -85,B 0,C 180,E1 -23956.844,E2 -23956.844} C_VEL
LIN {X 0,Y 153.997,Z 518.737,A -85,B 0,C 180,E1 -23958.717,E2 -23958.717} C_VEL
LIN {X 0,Y 154.993,Z 484.777,A -85,B 0,C 180,E1 -23961.793,E2 -23961.793} C_VEL
LIN {X 0,Y 155.076,Z 479.741,A -85,B 0,C 180,E1 -23962.394,E2 -23962.394} C_VEL
LIN {X 0,Y 155.31,Z 478.475,A -85,B 0,C 180,E1 -23962.973,E2 -23962.973} C_VEL
LIN {X 0,Y 156.344,Z 478.219,A -85,B 0,C 180,E1 -23963.864,E2 -23963.864} C_VEL
LIN {X 0,Y 161.565,Z 474.418,A -85,B 0,C 180,E1 -23965.785,E2 -23965.785} C_VEL
LIN {X 0,Y 163.88,Z 473.152,A -85,B 0,C 180,E1 -23966.764,E2 -23966.764} C_VEL
LIN {X 0,Y 166.84,Z 470.889,A -85,B 0,C 180,E1 -23967.605,E2 -23967.605} C_VEL
LIN {X 0,Y 170.787,Z 470.014,A -85,B 0,C 180,E1 -23969.592,E2 -23969.592} C_VEL
LIN {X 0,Y 172.903,Z 476.294,A -85,B 0,C 180,E1 -23973.281,E2 -23973.281} C_VEL
LIN {X 0,Y 175.023,Z 483.834,A -85,B 0,C 180,E1 -23977.037,E2 -23977.037} C_VEL
LIN {X 0,Y 176.194,Z 488.537,A -85,B 0,C 180,E1 -23979.186,E2 -23979.186} C_VEL
LIN {X 0,Y 181.75,Z 500.126,A -85,B 0,C 180,E1 -23981.972,E2 -23981.972} C_VEL
LIN {X 0,Y 184.021,Z 505.695,A -85,B 0,C 180,E1 -23983.064,E2 -23983.064} C_VEL
LIN {X 0,Y 185.809,Z 527.003,A -85,B 0,C 180,E1 -23984.808,E2 -23984.808} C_VEL
LIN {X 0,Y 186.564,Z 539.282,A -85,B 0,C 180,E1 -23985.693,E2 -23985.693} C_VEL
LIN {X 0,Y 182.573,Z 601.998,A -85,B 0,C 180,E1 -23987.898,E2 -23987.898} C_VEL
LIN {X 0,Y 180.823,Z 614.732,A -85,B 0,C 180,E1 -23988.644,E2 -23988.644} C_VEL
LIN {X 0,Y 178.616,Z 626.296,A -85,B 0,C 180,E1 -23989.702,E2 -23989.702} C_VEL
LIN {X 0,Y 175.542,Z 638.695,A -85,B 0,C 180,E1 -23991.277,E2 -23991.277} C_VEL
LIN {X 0,Y 172.346,Z 649.081,A -85,B 0,C 180,E1 -23993.024,E2 -23993.024} C_VEL
LIN {X 0,Y 168.47,Z 659.715,A -85,B 0,C 180,E1 -23995.362,E2 -23995.362} C_VEL
LIN {X 0,Y 164.898,Z 668.403,A -85,B 0,C 180,E1 -23997.809,E2 -23997.809} C_VEL
LIN {X 0,Y 160.807,Z 677.845,A -85,B 0,C 180,E1 -24001.266,E2 -24001.266} C_VEL
LIN {X 0,Y 157.12,Z 685.339,A -85,B 0,C 180,E1 -24004.854,E2 -24004.854} C_VEL
LIN {X 0,Y 153.919,Z 691.352,A -85,B 0,C 180,E1 -24008.575,E2 -24008.575} C_VEL
LIN {X 0,Y 151.49,Z 696.105,A -85,B 0,C 180,E1 -24012.45,E2 -24012.45} C_VEL
LIN {X 0,Y 149.683,Z 699.739,A -85,B 0,C 180,E1 -24016.423,E2 -24016.423} C_VEL
LIN {X 0,Y 148.794,Z 701.61,A -85,B 0,C 180,E1 -24019.11,E2 -24019.11} C_VEL
LIN {X 0,Y 148.173,Z 703.034,A -85,B 0,C 180,E1 -24021.82,E2 -24021.82} C_VEL
LIN {X 0,Y 147.797,Z 704.033,A -85,B 0,C 180,E1 -24024.543,E2 -24024.543} C_VEL
LIN {X 0,Y 147.597,Z 704.844,A -85,B 0,C 180,E1 -24029.387,E2 -24029.387} C_VEL
LIN {X 0,Y 147.614,Z 704.677,A -85,B 0,C 180,E1 -24032.729,E2 -24032.729} C_VEL
LIN {X 0,Y 147.774,Z 704.083,A -85,B 0,C 180,E1 -24035.459,E2 -24035.459} C_VEL
LIN {X 0,Y 148.121,Z 703.104,A -85,B 0,C 180,E1 -24038.184,E2 -24038.184} C_VEL
LIN {X 0,Y 148.726,Z 701.72,A -85,B 0,C 180,E1 -24040.896,E2 -24040.896} C_VEL
LIN {X 0,Y 150.132,Z 698.816,A -85,B 0,C 180,E1 -24044.92,E2 -24044.92} C_VEL
LIN {X 0,Y 152.101,Z 694.871,A -85,B 0,C 180,E1 -24048.872,E2 -24048.872} C_VEL
LIN {X 0,Y 154.862,Z 689.756,A -85,B 0,C 180,E1 -24052.691,E2 -24052.691} C_VEL
LIN {X 0,Y 158.155,Z 683.311,A -85,B 0,C 180,E1 -24056.384,E2 -24056.384} C_VEL
